// ---- POUs/StringHelper/cutStrNumberToSeperator.TcPOU
{attribute 'no_check'}
//Cut "number" from left site of string. Value will be written into LREAL Target variable in case found string is a valid number
//Function return value will be S_OK if a number is found, S_FALSE if string is empty and E_HRESULTADSERR.ERROR in case found characters are not a number
//Attention! do not use variables smaller then T_MaxString for Source parameter
FUNCTION cutStrNumberToSeperator : HRESULT
VAR_INPUT
	Seperator									:	STRING(5);
END_VAR
VAR_IN_OUT
	Source										:	T_MAXSTRING;
	Target										:	LREAL;
END_VAR
VAR
	tmpString									:	STRING;
	pSource										:	POINTER TO 	T_MAXSTRING;
END_VAR


	pSource										:= ADR(Source);
	tmpString									:= cutStrToSeperator(Seperator, pSource^);
	IF tmpString[0] = 0
	THEN
		cutStrNumberToSeperator					:= S_FALSE;				
	ELSIF isStringNumeric(ADR(tmpString)) 
	THEN 
		Target 									:= TO_LREAL(tmpString); 
	
		cutStrNumberToSeperator					:= S_OK;
	ELSE 
		cutStrNumberToSeperator					:= E_HRESULTADSERR.ERROR;
	END_IF

END_FUNCTION

// ---- POUs/StringHelper/STR_TO_ASC.TcPOU
FUNCTION STR_TO_ASC : BYTE
VAR_INPUT
	str : STRING;
END_VAR
VAR
	pChar : POINTER TO BYTE;
END_VAR

	pChar 		:= ADR(str);
	STR_TO_ASC 	:= pChar^;

END_FUNCTION

// ---- POUs/System/SystemInfo.TcPOU
{attribute 'no_check'}
//Provides all information of PlcAppSystemInfo plus addtional infos like time stamps from various source and in different formats
//
//PlcAppSystemInfo -> https://infosys.beckhoff.com/english.php?content=../content/1033/globaldatatypes/9007199969559691.html&id=7934476013631172214
//TwimCAT time sources -> https://infosys.beckhoff.com/english.php?content=../content/1033/ethercatsystem/2469114379.html&id=
//
FUNCTION_BLOCK SystemInfo
VAR_OUTPUT CONSTANT
{attribute 'displaymode':='binary'}
	OPTION_US_DATE_FORMAT									:	BYTE := 2#0000_0001; //Enable US date format in time stamp - mm/dd/yy
{attribute 'displaymode':='binary'}
	OPTION_US_TIME_FORMAT									:	BYTE := 2#0000_0010; //Enable time in US format - AM/PM vs 24h
{attribute 'displaymode':='binary'} 
	OPTION_TIME_STR_ADD_MS									:	BYTE := 2#0000_0100; //Add ms to time string 
{attribute 'displaymode':='binary'} 
	OPTION_DISABLE_DEV_IDENT								:	BYTE := 2#0000_1000; //Disable to read device identification during boot up (Call FB_GetDeviceIdentificationEx)
END_VAR                     								
VAR_INPUT                   						
	Enable													:	BOOL := TRUE; //Enable function block
	ResetTrig												:	BOOL := FALSE; //Reset Old boot data fault signal
	RtcSyncCylce											:	DWORD := 60; //in seconds - see documentation for "FB_LocalSystemTime"
	KeepOutputsOnBP 										: 	BOOL := FALSE; //The flag can be set to avoid that the outputs are zero-filled if a breakpoint is reached. The task keeps running. Only the execution of PLC code is interrupted.
{attribute 'displaymode':='binary'}
	Options													:	BYTE := 2#0000_0000; //option constants are alreay predefined, so they can accordingly be passed symbolically to the block 
	DateStrSeperator										:	STRING(1) := '/';
END_VAR
VAR_OUTPUT
//PlcAppSystemInfo and cycle time inforamtion from caller task 
	ObjId													: 	OTCID; //Object ID of the PLC project instance
	AdsPort 												: 	UINT; //ADS port of PLC application 
	TComSrvPtr 												: 	ITComObjectServer; // Pointer to TcCOM Object Server 
	AppName													: 	STRING(63); //TwinCAT generated name containing the port number. 
	ProjectName 											: 	STRING(63); //The name of the PLC project. 
	AppTimestampDT											:	DT; //Date and time of application start 
	AppTimestamp											:	STRING(25);	//Date and time of application start in string format
	TaskIndex												:	INT ; //Task index of SysInfo caller
	TaskCnt													: 	UDINT; //The number of tasks in the actual runtime system
	
	Flags 													: 	DWORD; //Boot flags
	LicensesPending 										: 	BOOL;
	BSODOccured 											: 	BOOL;										
	BootDataLoaded											: 	BOOL;//PERSISTENT variables: LOADED (without error)
	OldBootData												: 	BOOL; //PERSISTENT variables: INVALID (the back-up copy was loaded, since no valid data was present)
	NoBootDataLoaded										:	BOOL; //Error no boot data loaded
//	PersistentStatus 										: 	EPlcPersistentStatus;

	LoggedIn												:	BOOL;
	ShutdownInProgress 										: 	BOOL;	
	OnlineChangeCount										: 	UDINT; //The number of online changes made since the last complete download.
	OnlineChange											:	BOOL; //Online change count changed since last plc cycle

{attribute 'displaymode':='hex'}
	CpuCounter												:	ULINT;
	CycleTime         										: 	UDINT;//Cylce time read from PlcAppSystemInfo in multiples of 100 ns.
	CycleTimeNS         									: 	UDINT;//Cylce time in nanoseconds
	CycleTimeT       										: 	TIME; //Cycle time in time format
	CycleTimeLT       										: 	LTIME; //Cycle time in ltime format
	CycleTimeFloat											:	LREAL;//Cycle time in float format <s.ms>

	DevIdentValid											:	BOOL;
	pDevIdent												:	POINTER TO ST_DeviceIdentificationEx := ADR(InstGetDevIdent.stDevIdent);
	
//General	
	TimezoneId												: 	E_TimeZoneID;
	TimeZoneInfo											:	ST_TimeZoneInformation; //Provides actual time zone and bias from local time to UTC e.g. UTC=MEC-01:00 (-60min from lcoal MEZ in Standard time to UTC)
	MonthDays												:	WORD;
	LeapYear												:	BOOL;
	DayOfYear												:	WORD;
	WeekOfYear												:	WORD;
	UtcTimeFT												:	Tc2_Utilities.T_FILETIME; //Current UTC System/TwinCAT time T_FILETIME format, structure representing a 64-bit value with the a number of 100-nanosecond intervals since January 1, 1601 (UTC) (dwLowDateTime : DWORD / dwHighDateTime : DWORD)
//	UtcTimeFT												:	Tc2_Utilities.T_FILETIME64; //Current UTC System/TwinCAT time T_FILETIME format, structure representing a 64-bit value with the a number of 100-nanosecond intervals since January 1, 1601 (UTC) (dwLowDateTime : DWORD / dwHighDateTime : DWORD)
	UtcTimeSTRUCT											:	Tc2_Utilities.TIMESTRUCT; //Current UTC System/TwinCAT time in TIMESTRUCT format
	UtcTimezoneBias											:	DINT;   //Bias from UTC to local time in minutes e.g. MEZ=UTC+01:00 (60min)  
	TimeDT													:	DATE_AND_TIME;	//Current time in DATE_AND_TIME format: DT#1970-01-01-00:00 -> DT#2106-02-06-06:28:15
//	TimeLDT													:	LDATE_AND_TIME;	//Current time in 64bit LDATE_AND_TIME format: DT#1970-01-01-00:00 -> DT#2262-4-10-23:59:59.99999999
	TimeTOD													:	TOD; //Current time in TOD format, range from TOD#00:00 -> TOD#1193:02:47.295
	TimeFT													:	Tc2_Utilities.T_FILETIME; //Current time in T_FILETIME format, structur representing a 64-bit value with the a number of 100-nanosecond intervals since January 1, 1601 (UTC) (dwLowDateTime : DWORD / dwHighDateTime : DWORD)
//	TimeFT													:	Tc2_Utilities.T_FILETIME64; //Current time in T_FILETIME format, structur representing a 64-bit value with the a number of 100-nanosecond intervals since January 1, 1601 (UTC) (dwLowDateTime : DWORD / dwHighDateTime : DWORD)
	TimeSTRUCT												:	Tc2_Utilities.TIMESTRUCT; //Current time in TIMESTRUCT format
	Datestamp												:	DATE; //D#1970-01-01 -> D#2106-02-06
	DateStr													:	STRING(15);	(* dd.mm.jj or mm.dd.jj *)	
	TimeStr													:	STRING(15);	(* hh:mm:ss.xxx or hh:mm:ss.xxxPM/AM *)
	TimeStamp												:	STRING(25); (* DateStr + TimeStr *)	
	TimeStamp2												:	STRING(25); (* YYYY-MM-DDTHHMMSS for example YYYY-MM-DD_HHMMSS_Name.txt *)
	TimeStamp3												:	STRING(25); (* YYYY-MM-DD-hh:mm:ss.xxx *)
	DateStrISO												:	STRING(15);	(* jjjj-mm-dd *)
	TimeStrISO												:	STRING(15);	(* hh:mm:ss *)
	TimeStrISO2												:	STRING(15);	(* hh:mm:ss.xxx *)	
	TimeStampIso											:	STRING(30);	(* jjjj-mm-dd'T'hh:mm:ss.xxx local time*)	
//	TimeStampIsoZulu										:	STRING(30);	(* jjjj-mm-dd'T'hh:mm:ss.xmsZ - Iso timestamp in UTC (ZULU)*)	
//	TimeStampIsoUtc											:	STRING(30);	(* jjjj-mm-dd'T'hh:mm:ss.xms+mm:ss - Iso timestamp with UTC offset *)	

	TimeStampStartup										:	DATE_AND_TIME; //Timestamp of startup
	DCTime													:	Tc2_EtherCAT.T_DCTIME64; //Current TwinCAT distributed clock time in 64-bit T_DCTIME64 format. The smallest unit is a nanosecond.
	DCTimeSTRUCT											:	Tc2_Utilities.TIMESTRUCT;//Current TwinCAT distributed clock time in TIMESTRUCT format
//	SysTimeFT												:	Tc2_Utilities.T_FILETIME64; //Current UTC System/TwinCAT time T_FILETIME format, structure representing a 64-bit value with the a number of 100-nanosecond intervals since January 1, 1601 (UTC) (dwLowDateTime : DWORD / dwHighDateTime : DWORD)
	SysTimeFT												:	Tc2_Utilities.T_FILETIME; //Current UTC System/TwinCAT time T_FILETIME format, structure representing a 32-bit value since January 1, 1601 (UTC) (dwLowDateTime : DWORD / dwHighDateTime : DWORD)
	SysTimeSTRUCT											:	Tc2_Utilities.TIMESTRUCT; //Current UTC System/TwinCAT time in TIMESTRUCT format
	
END_VAR
VAR
	(* Inst. Get Taskindex *)
	InstGETCURTASKINDEX										: 	GETCURTASKINDEX;
	InstLocalSystemTime										:	FB_LocalSystemTime;
	InstNtSetLocalTime										:	NT_SetLocalTime := (NETID := '', TMOUT := DEFAULT_ADS_TIMEOUT);
	InstTimeZoneInfo										:	FB_GetTimeZoneInformation;
	InstCpuCouter											:	GETCPUCOUNTER;
	InstSystemTime											:	GetSystemTime;
	
	
	InstGetDevIdent											:	FB_GetDeviceIdentificationEx;
	_OnlineChangeCount										: 	UDINT; 
	_sec													:	WORD;
	_hour													:	WORD;
	_day													:	WORD;
	_Init													:	BOOL;
END_VAR

	(* Evaluate the PlcAppSystemInfo and and get sytstem timestamp					*)
	(********************************************************************************)
	
(* Get Current Task Index ************************************************************************)
	IF InstGETCURTASKINDEX.index = 0 then InstGETCURTASKINDEX(index => TaskIndex); END_IF

(* Read System Info Current Task *****************************************************************)	
	(* Get static information and boot error messages *)
	IF TwinCAT_SystemInfoVarList._TaskInfo[InstGETCURTASKINDEX.Index].FirstCycle 
	THEN
		AppTimestampDT										:= TwinCAT_SystemInfoVarList._AppInfo.AppTimestamp;
		AppTimestamp										:= DT_TO_STRING(AppTimestampDT);
		AppTimestamp										:= DELETE(AppTimestamp,3,1);
			
		TaskIndex											:= InstGETCURTASKINDEX.Index;
		TaskCnt 											:= TwinCAT_SystemInfoVarList._AppInfo.TaskCnt;
		
		ObjId												:= TwinCAT_SystemInfoVarList._AppInfo.ObjId;
		AppName												:= TwinCAT_SystemInfoVarList._AppInfo.AppName;	
		ProjectName											:= TwinCAT_SystemInfoVarList._AppInfo.ProjectName;	
		AdsPort												:= TwinCAT_SystemInfoVarList._AppInfo.AdsPort;	
			
		Flags												:= TwinCAT_SystemInfoVarList._AppInfo.Flags;
//		PersistentStatus									:= TwinCAT_SystemInfoVarList._AppInfo.PersistentStatus;
		
		BootDataLoaded										:= TwinCAT_SystemInfoVarList._AppInfo.BootDataLoaded;
		OldBootData											:= TwinCAT_SystemInfoVarList._AppInfo.OldBootData;
		NoBootDataLoaded									:= NOT BootDataLoaded AND NOT OldBootData;
		BSODOccured 										:= TwinCAT_SystemInfoVarList._AppInfo.BSODOccured;
		
		CycleTime         									:= TwinCAT_SystemInfoVarList._TaskInfo[TaskIndex].CycleTime;
		CycleTimeNS         								:= TwinCAT_SystemInfoVarList._TaskInfo[TaskIndex].CycleTime * 100;
		CycleTimeT											:= LREAL_TO_TIME(UDINT_TO_LREAL(CycleTime) * 0.0001 );
		CycleTimeLT											:= TO_LTIME(CycleTimeNS);	
		CycleTimeFloat										:= (UDINT_TO_LREAL(CycleTime) * 0.0001 / 1000.0);	
		
	ELSIF ResetTrig
	THEN
		resetBootInfo();
	ELSIF NOT Enable
	THEN
		RETURN;
	END_IF
	
	OnlineChangeCount										:= TwinCAT_SystemInfoVarList._AppInfo.OnlineChangeCnt;
	OnlineChange											:= _OnlineChangeCount <> OnlineChangeCount;
	_OnlineChangeCount										:= OnlineChangeCount;
	LoggedIn 												:= TwinCAT_SystemInfoVarList._AppInfo.LoggedIn;
	ShutdownInProgress 										:= TwinCAT_SystemInfoVarList._AppInfo.ShutdownInProgress;
	LicensesPending 										:= TwinCAT_SystemInfoVarList._AppInfo.LicensesPending;
	TComSrvPtr												:= TwinCAT_SystemInfoVarList._AppInfo.TComSrvPtr;
	TwinCAT_SystemInfoVarList._AppInfo.KeepOutputsOnBP		:= KeepOutputsOnBP;		

(* CPU System counter ****************************************************************************)
	InstCpuCouter(cpuCntLoDW => CpuCounter);	
	MEMCPY(ADR(CpuCounter) + SIZEOF(InstCpuCouter.cpuCntHiDW),ADR(InstCpuCouter.cpuCntHiDW),SIZEOF(InstCpuCouter.cpuCntHiDW));
	
(* Get device identification structure ***********************************************************)
	InstGetDevIdent(
		bExecute	:= NOT Options.3, 
		tTimeout	:= , 
		sNetId		:= , 
		bBusy		=> , 
		bError		=> , 
		nErrorID	=> , 
		stDevIdent	=> );	
	pDevIdent												:= ADR(InstGetDevIdent.stDevIdent);
	IF NOT InstGetDevIdent.bBusy
	THEN
		DevIdentValid										:= NOT InstGetDevIdent.bError;
		
		IF InstGetDevIdent.bError AND ResetTrig
		THEN
			InstGetDevIdent(bExecute := FALSE);			
		END_IF
	ELSE	
		DevIdentValid										:= FALSE;
	END_IF
	
(* Read timezone information every day time ******************************************************)
	IF Enable AND NOT InstTimeZoneInfo.bExecute
		OR InstTimeZoneInfo.bBusy
	THEN
		InstTimeZoneInfo(
			sNetID	:= , 
			bExecute:= TRUE, 
			tTimeout:= , 
			bBusy	=> , 
			bError	=> , 
			nErrID	=> , 
			tzID	=> TimeZoneId, 
			tzInfo	=> TimeZoneInfo);
		IF NOT InstTimeZoneInfo.bBusy 
		THEN
			CASE TimeZoneId OF 
			eTimeZoneID_Invalid:	UtcTimezoneBias			:= 0;				
			eTimeZoneID_Standard:	UtcTimezoneBias			:= -1 * (TimeZoneInfo.bias + TimeZoneInfo.standardBias);
			eTimeZoneID_Daylight:	UtcTimezoneBias			:= -1 * (TimeZoneInfo.bias + TimeZoneInfo.daylightBias);
			ELSE //eTimeZoneID_Unknown:		
				UtcTimezoneBias								:= 0;	
			END_CASE
		END_IF
	ELSIF NOT Enable AND InstTimeZoneInfo.bExecute 
		OR InstTimeZoneInfo.bError AND ResetTrig
	THEN
		InstTimeZoneInfo(bExecute:= FALSE);
	END_IF
		
(* Actual EtherCAT DC time in DCTIME64 format ****************************************************************)
	DCTime													:= F_GetActualDcTime64();
	DCTimeSTRUCT											:= DCTIME64_TO_SYSTEMTIME(DCTime);

(* Get TwinCAT/system time according to system time zone initialized during TC start ******************************************************)
	InstSystemTime(timeHiDW => UtcTimeFT.dwHighDateTime,timeLoDW => UtcTimeFT.dwLowDateTime );
	SysTimeSTRUCT											:= FILETIME_TO_SYSTEMTIME(UTCTimeFT);	
	
//	SysTimeFT												:= F_GetSystemTime();	 
//	SysTimeSTRUCT											:= FILETIME64_TO_SYSTEMTIME(UTCTimeFT);	 
	
(* evalutate systemtime ************************************************************************)
	InstLocalSystemTime(
		sNetID		:= '',
		bEnable		:= Enable,
		dwCycle		:= SEL(InstNtSetLocalTime.START, RtcSyncCylce, 1), //Short update cylce to read windows time after it was set
		dwopt		:= (* Default *),
		tTimeout	:= (* Default *),
		bValid		=> ,
		systemTime	=> TimeSTRUCT,
		tzID		=> );

(* Get TwinCAT/system time in UTC Filetime format ******************************************************)
	IF InstLocalSystemTime.bValid 
	THEN				
		//Update cyclic
//		TimeFT												:= SYSTEMTIME_TO_FILETIME64(TimeSTRUCT);
		TimeFT												:= SYSTEMTIME_TO_FILETIME(TimeSTRUCT);
		TimeDT 												:= SYSTEMTIME_TO_DT(TimeSTRUCT);
//		TimeLDT												:= SYSTEMTIME_TO_LDT(TimeSTRUCT);	
		TimeStamp3											:= SYSTEMTIME_TO_STRING(TimeSTRUCT);
		TimeTOD												:= SEL(Options.2 ,TO_TOD(TimeDT)  , DWORD_TO_TOD(TO_DWORD(TO_TOD(TimeDT)) + TimeSTRUCT.wMilliseconds));  
		TimeStrISO											:= DELETE(TO_STRING(TimeTOD),4,1);

		IF TimeSTRUCT.wMilliseconds < 10 
		THEN
			TimeStrISO2 									:= CONCAT(TimeStrISO,CONCAT('.00',WORD_TO_STRING(TimeSTRUCT.wMilliseconds)));
		ELSIF TimeSTRUCT.wMilliseconds < 100
		THEN
			TimeStrISO2 									:= CONCAT(TimeStrISO,CONCAT('.0',WORD_TO_STRING(TimeSTRUCT.wMilliseconds)));			
		ELSE        										
			TimeStrISO2 									:= CONCAT(TimeStrISO,CONCAT('.',WORD_TO_STRING(TimeSTRUCT.wMilliseconds)));	
		END_IF 	
		
		TimeStampISO										:= CONCAT(DateStrISO , CONCAT('T',TimeStrISO2));
				
		UtcTimeFT											:= F_TranslateFileTimeBias(TimeFT,UtcTimezoneBias,TRUE);
		UtcTimeSTRUCT										:= FILETIME_TO_SYSTEMTIME(UTCTimeFT);	
//		UtcTimeFT											:= F_TranslateFileTime64Bias(TimeFT,UtcTimezoneBias,TRUE);
//		UtcTimeSTRUCT										:= FILETIME64_TO_SYSTEMTIME(UTCTimeFT);	

//		TimeStampIsoZulu									:= SYSTEMTIME_TO_ISO8601(UtcTimeSTRUCT,0,FALSE,3);
//		TimeStampIsoZulu									:= CONCAT(DELETE(TimeStampIsoZulu,6,24),'Z');
//		TimeStampIsoUtc										:= SYSTEMTIME_TO_ISO8601(UtcTimeSTRUCT,TO_INT(UtcTimezoneBias),TRUE,3);
	
		//Create time format
		IF Options.1
		THEN (* US time format hh.mm.ss AM/PM ***************)
			IF TimeSTRUCT.wHour < 10 
			THEN
				TimeStr 									:= CONCAT('0',WORD_TO_STRING(TimeSTRUCT.wHour));
			ELSIF TimeSTRUCT.wHour > 12 
			THEN
				TimeStr 									:= WORD_TO_STRING(TimeSTRUCT.wHour - 12);
				IF TimeSTRUCT.wHour - 12 < 10
				THEN
					TimeStr									:= CONCAT('0',TimeStr);
				END_IF
			ELSE         									
				TimeStr 									:= WORD_TO_STRING(TimeSTRUCT.wHour);
			END_IF		                                    
		ELSE  (* Time hh.mm.ss.xxms ***************)          
			IF TimeSTRUCT.wHour < 10                        
			THEN                                            
				TimeStr 									:= CONCAT('0',WORD_TO_STRING(TimeSTRUCT.wHour));
			ELSE        									
				TimeStr 									:= WORD_TO_STRING(TimeSTRUCT.wHour);
			END_IF			
		END_IF
		
		TimeStr 											:= CONCAT(TimeStr,':');
		
		IF TimeSTRUCT.wMinute < 10 
		THEN
			TimeStr 										:= CONCAT(TimeStr,CONCAT('0',WORD_TO_STRING(TimeSTRUCT.wMinute)));
		ELSE
			TimeStr 										:= CONCAT(TimeStr,WORD_TO_STRING(TimeSTRUCT.wMinute));
		END_IF
		
		TimeStr 											:= CONCAT(TimeStr,':');
		
		IF TimeSTRUCT.wSecond < 10 
		THEN
			TimeStr 										:= CONCAT(TimeStr,CONCAT('0',WORD_TO_STRING(TimeSTRUCT.wSecond)));
		ELSE        										
			TimeStr 										:= CONCAT(TimeStr,WORD_TO_STRING(TimeSTRUCT.wSecond));
		END_IF  
												
		IF Options.2
		THEN //add ms to timestamp
			TimeStr 										:= CONCAT(TimeStr,'.');
			TimeStr 										:= CONCAT(TimeStr,WORD_TO_STRING(TimeSTRUCT.wMilliseconds));
		END_IF
		
		IF Options.1
		THEN //US time format
			TimeStr 										:= CONCAT(TimeStr,SEL(TimeSTRUCT.wHour > 12,' AM', ' PM'));
		END_IF
		
		(* TimeStamp Format DE: DD.MM.YY-Stunde:Minute:Sekunde.xxx,*)
		TimeStamp 											:= CONCAT(DateStr,'-');
		TimeStamp 											:= CONCAT(TimeStamp,TimeStr);
		
		IF _hour <> TimeSTRUCT.wHour OR NOT _Init
		THEN
			_Hour											:= TimeSTRUCT.wHour;		
			//Create date in US fromat with seperator / ************************************************
			IF Options.0
			THEN (* Date mm/dd/jj ********************)
				IF TimeSTRUCT.wMonth < 10 
				THEN
					DateStr 								:= CONCAT('0',WORD_TO_STRING(TimeSTRUCT.wMonth));
				ELSE        								
					DateStr 								:= WORD_TO_STRING(TimeSTRUCT.wMonth);
				END_IF		                                
				DateStr 									:= CONCAT(DateStr,DateStrSeperator);
				IF TimeSTRUCT.wDay < 10                     
				THEN                                        
					DateStr 								:= CONCAT(DateStr,CONCAT('0',WORD_TO_STRING(TimeSTRUCT.wDay)));
				ELSE        								
					DateStr 								:= CONCAT(DateStr,WORD_TO_STRING(TimeSTRUCT.wDay));
				END_IF                                      
															
				DateStr 									:= CONCAT(DateStr,DateStrSeperator);
				DateStr 									:= CONCAT(DateStr,RIGHT(WORD_TO_STRING(TimeSTRUCT.wYear),2));		
		                                                    
			ELSE (* Date dd.mm.jj ********************)	    
				IF TimeSTRUCT.wDay < 10                     
				THEN                                        
					DateStr 								:= CONCAT('0',WORD_TO_STRING(TimeSTRUCT.wDay));
				ELSE        								
					DateStr 								:= WORD_TO_STRING(TimeSTRUCT.wDay);
				END_IF                                      
				DateStr 									:= CONCAT(DateStr,DateStrSeperator);
				IF TimeSTRUCT.wMonth < 10                   
				THEN                                        
					DateStr 								:= CONCAT(DateStr,CONCAT('0',WORD_TO_STRING(TimeSTRUCT.wMonth)));
				ELSE        								
					DateStr 								:= CONCAT(DateStr,WORD_TO_STRING(TimeSTRUCT.wMonth));
				END_IF                                      
															
				DateStr 									:= CONCAT(DateStr,DateStrSeperator);
				DateStr 									:= CONCAT(DateStr,RIGHT(WORD_TO_STRING(TimeSTRUCT.wYear),2));	
			END_IF      

			DateStrISO										:= DELETE(TO_STRING(TO_DATE(TimeDT)),2,1);
			
			(* information of year *)                       
			MonthDays										:= F_GetMaxMonthDays(TimeSTRUCT.wYear,TimeSTRUCT.wMonth);
			LeapYear										:= F_YearIsLeapYear(TimeSTRUCT.wYear) ;
			WeekOfYear										:= F_GetWeekOfTheYear(TimeDT);
			DayOfYear										:= F_GetDOYOfYearMonthDay(TimeSTRUCT.wYear,TimeSTRUCT.wMonth,TimeSTRUCT.wDay);
			DateStamp										:= TO_DATE(TimeDT);		
			
			IF NOT _INIT AND_THEN TO_DINT(TimeStampStartup) = 0  
			THEN					
				TimeStampStartup							:= SYSTEMTIME_TO_DT(TimeSTRUCT);
			END_IF
			
			IF NOT InstTimeZoneInfo.bBusy THEN InstTimeZoneInfo(bExecute:= FALSE); END_IF

            _INIT											:= TRUE;            
		END_IF //hour
		
		IF _sec <> TimeSTRUCT.wSecond 
		THEN	
			_sec 											:= TimeSTRUCT.wSecond;
														
			(* TimeStamp2 FileName YYYY-MM-DD_HHMMSS *)
			TimeStamp2										:= CONCAT(DateStrISO , '_');
			IF TimeSTRUCT.wHour < 10                    	
			THEN                                        	
				TimeStamp2 									:= CONCAT(TimeStamp2,CONCAT('0',WORD_TO_STRING(TimeSTRUCT.wHour)));
			ELSE           									
				TimeStamp2 									:= CONCAT(TimeStamp2,WORD_TO_STRING(TimeSTRUCT.wHour));
			END_IF                                      	
			IF TimeSTRUCT.wMinute < 10                  	
			THEN                                        	
				TimeStamp2 									:= CONCAT(TimeStamp2,CONCAT('0',WORD_TO_STRING(TimeSTRUCT.wMinute)));
			ELSE           									
				TimeStamp2 									:= CONCAT(TimeStamp2,WORD_TO_STRING(TimeSTRUCT.wMinute));
			END_IF                                      	
			IF TimeSTRUCT.wSecond < 10                  	
			THEN                                        	
				TimeStamp2 									:= CONCAT(TimeStamp2,CONCAT('0',WORD_TO_STRING(TimeSTRUCT.wSecond)));
			ELSE           									
				TimeStamp2 									:= CONCAT(TimeStamp2,WORD_TO_STRING(TimeSTRUCT.wSecond));
			END_IF
		END_IF //second update
													
	END_IF

(* set system time *****************************************************************************)
	InstNtSetLocalTime(
		NETID		:= , 
		TIMESTR		:= , 
		START		:= , // Start by Methode "SetSysTime" 
		TMOUT		:= , 
		BUSY		=> , 
		ERR			=> ); 
	
	IF InstNtSetLocalTime.START AND NOT InstNtSetLocalTime.BUSY
	THEN //Take care that all timestamp get updated after set a new time
		InstNtSetLocalTime.START							:= FALSE;	
		_Init												:= FALSE;								
	END_IF
	
(**************************************************************************************************)

PROPERTY PUBLIC actDCTimeWithTimezoneBias : T_DCTIME64
GET
actDCTimeWithTimezoneBias							:= F_GetActualDcTime64() + (TO_ULINT(UtcTimezoneBias) * 60 * EC_DCTIME_TICKSPERSEC64);
END_GET
END_PROPERTY

PROPERTY PUBLIC optAddmsToTimeString : BOOL
GET
optAddmsToTimeString := Options.2;
END_GET
SET
Options.2 := optAddmsToTimeString;
END_SET
END_PROPERTY

PROPERTY PUBLIC  optDisableReadDeviceIdentification : BOOL
GET
optDisableReadDeviceIdentification := Options.3;
END_GET
SET
Options.3 := optDisableReadDeviceIdentification;
END_SET
END_PROPERTY

PROPERTY PUBLIC optEnableUSDateFormat : BOOL
GET
optEnableUSDateFormat := Options.0;
END_GET
SET
Options.0 := optEnableUSDateFormat;
END_SET
END_PROPERTY

PROPERTY PUBLIC optEnableUSTimeFormat : BOOL
GET
optEnableUSTimeFormat := Options.1;
END_GET
SET
Options.1 := optEnableUSTimeFormat;
END_SET
END_PROPERTY

METHOD PUBLIC resetBootInfo : BOOL  //Return value = TRUE if execution finished
VAR_INPUT
END_VAR
OldBootData 												:= FALSE;
BSODOccured													:= FALSE;
NoBootDataLoaded											:= FALSE;
resetBootInfo												:= TRUE;
END_METHOD

METHOD PUBLIC setSysTime  : BOOL //Return value = TRUE if execution finished
VAR_INPUT
	TimeStruct		: TIMESTRUCT;
END_VAR
InstNtSetLocalTime(
		NETID		:= '', 
		TIMESTR		:= TimeStruct, 
		START		:= NOT InstNtSetLocalTime.START AND TimeStruct.wYear > 2000 
						AND TimeStruct.wDay > 0 AND TimeStruct.wMonth	< 32	
						AND TimeStruct.wMonth > 0 AND TimeStruct.wMonth	< 13	
						AND TimeStruct.wHour >= 0 AND TimeStruct.wHour	< 24	
						AND TimeStruct.wMinute >= 0 AND TimeStruct.wMinute < 60
						AND TimeStruct.wSecond >= 0 AND TimeStruct.wSecond < 60				
						OR InstNtSetLocalTime.BUSY, 
		TMOUT		:= , 
		BUSY		=> , 
		ERR			=> , 
		ERRID		=> );
		
setSysTime													:= InstNtSetLocalTime.BUSY;
END_METHOD

END_FUNCTION_BLOCK

// ---- POUs/System/SystemInfo64.TcPOU
{attribute 'no_check'}
//Provides all information of PlcAppSystemInfo plus addtional infos like time stamps from various source and in different formats
//
//PlcAppSystemInfo -> https://infosys.beckhoff.com/english.php?content=../content/1033/globaldatatypes/9007199969559691.html&id=7934476013631172214
//TwimCAT time sources -> https://infosys.beckhoff.com/english.php?content=../content/1033/ethercatsystem/2469114379.html&id=
//
FUNCTION_BLOCK SystemInfo64
VAR_OUTPUT CONSTANT
{attribute 'displaymode':='binary'}
	OPTION_US_DATE_FORMAT									:	BYTE := 2#0000_0001; //Enable US date format in time stamp - mm/dd/yy
{attribute 'displaymode':='binary'}
	OPTION_US_TIME_FORMAT									:	BYTE := 2#0000_0010; //Enable time in US format - AM/PM vs 24h
{attribute 'displaymode':='binary'} 
	OPTION_TIME_STR_ADD_MS									:	BYTE := 2#0000_0100; //Add ms to time string 
{attribute 'displaymode':='binary'} 
	OPTION_DISABLE_DEV_IDENT								:	BYTE := 2#0000_1000; //Disable to read device identification during boot up (Call FB_GetDeviceIdentificationEx)
END_VAR                     								
VAR_INPUT                   						
	Enable													:	BOOL := TRUE; //Enable function block
	ResetTrig												:	BOOL := FALSE; //Reset Old boot data fault signal
	RtcSyncCylce											:	DWORD := 60; //in seconds - see documentation for "FB_LocalSystemTime"
	KeepOutputsOnBP 										: 	BOOL := FALSE; //The flag can be set to avoid that the outputs are zero-filled if a breakpoint is reached. The task keeps running. Only the execution of PLC code is interrupted.
{attribute 'displaymode':='binary'}
	Options													:	BYTE := 2#0000_0000; //option constants are alreay predefined, so they can accordingly be passed symbolically to the block 
	DateStrSeperator										:	STRING(1) := '/';
END_VAR
VAR_OUTPUT
//PlcAppSystemInfo and cycle time inforamtion from caller task 
	ObjId													: 	OTCID; //Object ID of the PLC project instance
	AdsPort 												: 	UINT; //ADS port of PLC application 
	TComSrvPtr 												: 	ITComObjectServer; // Pointer to TcCOM Object Server 
	AppName													: 	STRING(63); //TwinCAT generated name containing the port number. 
	ProjectName 											: 	STRING(63); //The name of the PLC project. 
	AppTimestampDT											:	DT; //Date and time of application start 
	AppTimestamp											:	STRING(25);	//Date and time of application start in string format
	TaskIndex												:	INT ; //Task index of SysInfo caller
	TaskCnt													: 	UDINT; //The number of tasks in the actual runtime system
	
	Flags 													: 	DWORD; //Boot flags
	LicensesPending 										: 	BOOL;
	BSODOccured 											: 	BOOL;										
	BootDataLoaded											: 	BOOL;//PERSISTENT variables: LOADED (without error)
	OldBootData												: 	BOOL; //PERSISTENT variables: INVALID (the back-up copy was loaded, since no valid data was present)
	NoBootDataLoaded										:	BOOL; //Error no boot data loaded
//	PersistentStatus 										: 	EPlcPersistentStatus;

	LoggedIn												:	BOOL;
	ShutdownInProgress 										: 	BOOL;	
	OnlineChangeCount										: 	UDINT; //The number of online changes made since the last complete download.
	OnlineChange											:	BOOL; //Online change count changed since last plc cycle

{attribute 'displaymode':='hex'}
	CpuCounter												:	ULINT;
	CycleTime         										: 	UDINT;//Cylce time read from PlcAppSystemInfo in multiples of 100 ns.
	CycleTimeNS         									: 	UDINT;//Cylce time in nanoseconds
	CycleTimeT       										: 	TIME; //Cycle time in time format
	CycleTimeLT       										: 	LTIME; //Cycle time in ltime format
	CycleTimeFloat											:	LREAL;//Cycle time in float format <s.ms>

	DevIdentValid											:	BOOL;
	pDevIdent												:	POINTER TO ST_DeviceIdentificationEx := ADR(InstGetDevIdent.stDevIdent);
	
//General	
	TimezoneId												: 	E_TimeZoneID;
	TimeZoneInfo											:	ST_TimeZoneInformation;
	MonthDays												:	WORD;
	LeapYear												:	BOOL;
	DayOfYear												:	WORD;
	WeekOfYear												:	WORD;
	UtcTimeFT												:	Tc2_Utilities.T_FILETIME64; //Current UTC System/TwinCAT time T_FILETIME format, structure representing a 64-bit value with the a number of 100-nanosecond intervals since January 1, 1601 (UTC) (dwLowDateTime : DWORD / dwHighDateTime : DWORD)
	UtcTimeSTRUCT											:	Tc2_Utilities.TIMESTRUCT; //Current UTC System/TwinCAT time in TIMESTRUCT format
	UtcTimezoneBias											:	DINT;   //Total timezone bias in minutes to UTC 
	TimeDT													:	DATE_AND_TIME;	//Current time in DATE_AND_TIME format: DT#1970-01-01-00:00 -> DT#2106-02-06-06:28:15
//	TimeLDT													:	LDATE_AND_TIME;	//Current time in 64bit LDATE_AND_TIME format: DT#1970-01-01-00:00 -> DT#2262-4-10-23:59:59.99999999
	TimeTOD													:	TOD; //Current time in TOD format, range from TOD#00:00 -> TOD#1193:02:47.295
	TimeFT													:	Tc2_Utilities.T_FILETIME64; //Current time in T_FILETIME format, structur representing a 64-bit value with the a number of 100-nanosecond intervals since January 1, 1601 (UTC) (dwLowDateTime : DWORD / dwHighDateTime : DWORD)
	TimeSTRUCT												:	Tc2_Utilities.TIMESTRUCT; //Current time in TIMESTRUCT format
	Datestamp												:	DATE; //D#1970-01-01 -> D#2106-02-06
	DateStr													:	STRING(15);	(* dd.mm.jj or mm.dd.jj *)	
	TimeStr													:	STRING(15);	(* hh:mm:ss.xxx or hh:mm:ss.xxxPM/AM *)
	TimeStamp												:	STRING(25); (* DateStr + TimeStr *)	
	TimeStamp2												:	STRING(25); (* YYYY-MM-DDTHHMMSS for example YYYY-MM-DD_HHMMSS_Name.txt *)
	TimeStamp3												:	STRING(25); (* YYYY-MM-DD-hh:mm:ss.xxx *)
	DateStrISO												:	STRING(15);	(* jj-mm-dd *)
	TimeStrISO												:	STRING(15);	(* hh:mm:ss *)
	TimeStampISO											:	STRING(25);	(* jj-mm-dd'T'hh:mm:ss.xxms *)	
	TimeStampStartup										:	DATE_AND_TIME; //Timestamp of startup
	DCTime													:	Tc2_EtherCAT.T_DCTIME64; //Current TwinCAT distributed clock time in 64-bit T_DCTIME64 format. The smallest unit is a nanosecond.
	DCTimeSTRUCT											:	Tc2_Utilities.TIMESTRUCT;//Current TwinCAT distributed clock time in TIMESTRUCT format
	SysTimeFT												:	Tc2_Utilities.T_FILETIME64; //Current UTC System/TwinCAT time T_FILETIME format, structure representing a 64-bit value with the a number of 100-nanosecond intervals since January 1, 1601 (UTC) (dwLowDateTime : DWORD / dwHighDateTime : DWORD)
	SysTimeSTRUCT											:	Tc2_Utilities.TIMESTRUCT; //Current UTC System/TwinCAT time in TIMESTRUCT format
	
END_VAR
VAR
	(* Inst. Get Taskindex *)
	InstGETCURTASKINDEX										: 	GETCURTASKINDEX;
	InstLocalSystemTime										:	FB_LocalSystemTime;
	InstNtSetLocalTime										:	NT_SetLocalTime := (NETID := '', TMOUT := DEFAULT_ADS_TIMEOUT);
	InstTimeZoneInfo										:	FB_GetTimeZoneInformation;
	InstCpuCouter											:	GETCPUCOUNTER;
	
	InstGetDevIdent											:	FB_GetDeviceIdentificationEx;
	_OnlineChangeCount										: 	UDINT; 
	_sec													:	WORD;
	_hour													:	WORD;
	_day													:	WORD;
	_Init													:	BOOL;
END_VAR

	(* Evaluate the PlcAppSystemInfo and and get sytstem timestamp					*)
	(********************************************************************************)
	
(* Get Current Task Index ************************************************************************)
	IF InstGETCURTASKINDEX.index = 0 then InstGETCURTASKINDEX(index => TaskIndex); END_IF

(* Read System Info Current Task *****************************************************************)	
	(* Get static information and boot error messages *)
	IF TwinCAT_SystemInfoVarList._TaskInfo[InstGETCURTASKINDEX.Index].FirstCycle 
	THEN
		AppTimestampDT										:= TwinCAT_SystemInfoVarList._AppInfo.AppTimestamp;
		AppTimestamp										:= DT_TO_STRING(AppTimestampDT);
		AppTimestamp										:= DELETE(AppTimestamp,3,1);
			
		TaskIndex											:= InstGETCURTASKINDEX.Index;
		TaskCnt 											:= TwinCAT_SystemInfoVarList._AppInfo.TaskCnt;
		
		ObjId												:= TwinCAT_SystemInfoVarList._AppInfo.ObjId;
		AppName												:= TwinCAT_SystemInfoVarList._AppInfo.AppName;	
		ProjectName											:= TwinCAT_SystemInfoVarList._AppInfo.ProjectName;	
		AdsPort												:= TwinCAT_SystemInfoVarList._AppInfo.AdsPort;	
			
		Flags												:= TwinCAT_SystemInfoVarList._AppInfo.Flags;
//		PersistentStatus									:= TwinCAT_SystemInfoVarList._AppInfo.PersistentStatus;
		
		BootDataLoaded										:= TwinCAT_SystemInfoVarList._AppInfo.BootDataLoaded;
		OldBootData											:= TwinCAT_SystemInfoVarList._AppInfo.OldBootData;
		NoBootDataLoaded									:= NOT BootDataLoaded AND NOT OldBootData;
		BSODOccured 										:= TwinCAT_SystemInfoVarList._AppInfo.BSODOccured;
		
		CycleTime         									:= TwinCAT_SystemInfoVarList._TaskInfo[TaskIndex].CycleTime;
		CycleTimeNS         								:= TwinCAT_SystemInfoVarList._TaskInfo[TaskIndex].CycleTime * 100;
		CycleTimeT											:= LREAL_TO_TIME(UDINT_TO_LREAL(CycleTime) * 0.0001 );
		CycleTimeLT											:= TO_LTIME(CycleTimeNS);	
		CycleTimeFloat										:= (UDINT_TO_LREAL(CycleTime) * 0.0001 / 1000.0);	
		
	ELSIF ResetTrig
	THEN
		resetBootInfo();
	ELSIF NOT Enable
	THEN
		RETURN;
	END_IF
	
	OnlineChangeCount										:= TwinCAT_SystemInfoVarList._AppInfo.OnlineChangeCnt;
	OnlineChange											:= _OnlineChangeCount <> OnlineChangeCount;
	_OnlineChangeCount										:= OnlineChangeCount;
	LoggedIn 												:= TwinCAT_SystemInfoVarList._AppInfo.LoggedIn;
	ShutdownInProgress 										:= TwinCAT_SystemInfoVarList._AppInfo.ShutdownInProgress;
	LicensesPending 										:= TwinCAT_SystemInfoVarList._AppInfo.LicensesPending;
	TComSrvPtr												:= TwinCAT_SystemInfoVarList._AppInfo.TComSrvPtr;
	TwinCAT_SystemInfoVarList._AppInfo.KeepOutputsOnBP		:= KeepOutputsOnBP;		

(* CPU System counter ****************************************************************************)
	InstCpuCouter(cpuCntLoDW => CpuCounter);	
	MEMCPY(ADR(CpuCounter) + SIZEOF(InstCpuCouter.cpuCntHiDW),ADR(InstCpuCouter.cpuCntHiDW),SIZEOF(InstCpuCouter.cpuCntHiDW));
	
(* Get device identification structure ***********************************************************)
	InstGetDevIdent(
		bExecute	:= NOT Options.3, 
		tTimeout	:= , 
		sNetId		:= , 
		bBusy		=> , 
		bError		=> , 
		nErrorID	=> , 
		stDevIdent	=> );	
	pDevIdent												:= ADR(InstGetDevIdent.stDevIdent);
	IF NOT InstGetDevIdent.bBusy
	THEN
		DevIdentValid										:= NOT InstGetDevIdent.bError;
		
		IF InstGetDevIdent.bError AND ResetTrig
		THEN
			InstGetDevIdent(bExecute := FALSE);			
		END_IF
	ELSE	
		DevIdentValid										:= FALSE;
	END_IF
	
(* Read timezone information every day time ******************************************************)
	IF Enable AND NOT InstTimeZoneInfo.bExecute
		OR InstTimeZoneInfo.bBusy
	THEN
		InstTimeZoneInfo(
			sNetID	:= , 
			bExecute:= TRUE, 
			tTimeout:= , 
			bBusy	=> , 
			bError	=> , 
			nErrID	=> , 
			tzID	=> TimeZoneId, 
			tzInfo	=> TimeZoneInfo);
		IF NOT InstTimeZoneInfo.bBusy 
		THEN
			CASE TimeZoneId OF 
			eTimeZoneID_Invalid:	UtcTimezoneBias			:= 0;				
			eTimeZoneID_Standard:	UtcTimezoneBias			:= -1 * (TimeZoneInfo.bias);
			eTimeZoneID_Daylight:	UtcTimezoneBias			:= -1 * (TimeZoneInfo.bias + TimeZoneInfo.daylightBias);
			ELSE //eTimeZoneID_Unknown:		
				UtcTimezoneBias								:= 0;	
			END_CASE
		END_IF
	ELSIF NOT Enable AND InstTimeZoneInfo.bExecute 
		OR InstTimeZoneInfo.bError AND ResetTrig
	THEN
		InstTimeZoneInfo(bExecute:= FALSE);
	END_IF
		
(* Actual EtherCAT DC time in DCTIME64 format ****************************************************************)
	DCTime													:= F_GetActualDcTime64();
	DCTimeSTRUCT											:= DCTIME64_TO_SYSTEMTIME(DCTime);

(* Get TwinCAT/system time according to system time zone initialized during TC start ******************************************************)
	SysTimeFT												:= F_GetSystemTime();	 
	SysTimeSTRUCT											:= FILETIME64_TO_SYSTEMTIME(UTCTimeFT);	 
	
(* evalutate systemtime ************************************************************************)
	InstLocalSystemTime(
		sNetID		:= '',
		bEnable		:= Enable,
		dwCycle		:= SEL(InstNtSetLocalTime.START, RtcSyncCylce, 1), //Short update cylce to read windows time after it was set
		dwopt		:= (* Default *),
		tTimeout	:= (* Default *),
		bValid		=> ,
		systemTime	=> TimeSTRUCT,
		tzID		=> );

(* Get TwinCAT/system time in UTC Filetime format ******************************************************)
	IF InstLocalSystemTime.bValid 
	THEN				
		//Update cyclic
		TimeFT												:= SYSTEMTIME_TO_FILETIME64(TimeSTRUCT);
		TimeDT 												:= SYSTEMTIME_TO_DT(TimeSTRUCT);
//		TimeLDT												:= SYSTEMTIME_TO_LDT(TimeSTRUCT);	
		TimeStamp3											:= SYSTEMTIME_TO_STRING(TimeSTRUCT);
		TimeTOD												:= SEL(Options.2 ,TO_TOD(TimeDT)  , DWORD_TO_TOD(TO_DWORD(TO_TOD(TimeDT)) + TimeSTRUCT.wMilliseconds));  
		TimeStrISO											:= DELETE(TO_STRING(TimeTOD),4,1);
		TimeStampISO										:= CONCAT(DateStrISO , CONCAT('T',TimeStrISO));
		
		UtcTimeFT											:= F_TranslateFileTime64Bias(TimeFT,UtcTimezoneBias,TRUE);
		UtcTimeSTRUCT										:= FILETIME64_TO_SYSTEMTIME(UTCTimeFT);	
	
		//Create time format
		IF Options.1
		THEN (* US time format hh.mm.ss AM/PM ***************)
			IF TimeSTRUCT.wHour < 10 
			THEN
				TimeStr 									:= CONCAT('0',WORD_TO_STRING(TimeSTRUCT.wHour));
			ELSIF TimeSTRUCT.wHour > 12 
			THEN
				TimeStr 									:= WORD_TO_STRING(TimeSTRUCT.wHour - 12);
				IF TimeSTRUCT.wHour - 12 < 10
				THEN
					TimeStr									:= CONCAT('0',TimeStr);
				END_IF
			ELSE         									
				TimeStr 									:= WORD_TO_STRING(TimeSTRUCT.wHour);
			END_IF		                                    
		ELSE  (* Time hh.mm.ss.xxms ***************)          
			IF TimeSTRUCT.wHour < 10                        
			THEN                                            
				TimeStr 									:= CONCAT('0',WORD_TO_STRING(TimeSTRUCT.wHour));
			ELSE        									
				TimeStr 									:= WORD_TO_STRING(TimeSTRUCT.wHour);
			END_IF			
		END_IF
		
		TimeStr 											:= CONCAT(TimeStr,':');
		
		IF TimeSTRUCT.wMinute < 10 
		THEN
			TimeStr 										:= CONCAT(TimeStr,CONCAT('0',WORD_TO_STRING(TimeSTRUCT.wMinute)));
		ELSE
			TimeStr 										:= CONCAT(TimeStr,WORD_TO_STRING(TimeSTRUCT.wMinute));
		END_IF
		
		TimeStr 											:= CONCAT(TimeStr,':');
		
		IF TimeSTRUCT.wSecond < 10 
		THEN
			TimeStr 										:= CONCAT(TimeStr,CONCAT('0',WORD_TO_STRING(TimeSTRUCT.wSecond)));
		ELSE        										
			TimeStr 										:= CONCAT(TimeStr,WORD_TO_STRING(TimeSTRUCT.wSecond));
		END_IF  
												
		IF Options.2
		THEN //add ms to timestamp
			TimeStr 										:= CONCAT(TimeStr,'.');
			TimeStr 										:= CONCAT(TimeStr,WORD_TO_STRING(TimeSTRUCT.wMilliseconds));
		END_IF
		
		IF Options.1
		THEN //US time format
			TimeStr 										:= CONCAT(TimeStr,SEL(TimeSTRUCT.wHour > 12,' AM', ' PM'));
		END_IF
		
		(* TimeStamp Format DE: DD.MM.YY-Stunde:Minute:Sekunde.xxx,*)
		TimeStamp 											:= CONCAT(DateStr,'-');
		TimeStamp 											:= CONCAT(TimeStamp,TimeStr);
		
		IF _hour <> TimeSTRUCT.wHour OR NOT _Init
		THEN
			_Hour											:= TimeSTRUCT.wHour;		
			//Create date in US fromat with seperator / ************************************************
			IF Options.0
			THEN (* Date mm/dd/jj ********************)
				IF TimeSTRUCT.wMonth < 10 
				THEN
					DateStr 								:= CONCAT('0',WORD_TO_STRING(TimeSTRUCT.wMonth));
				ELSE        								
					DateStr 								:= WORD_TO_STRING(TimeSTRUCT.wMonth);
				END_IF		                                
				DateStr 									:= CONCAT(DateStr,DateStrSeperator);
				IF TimeSTRUCT.wDay < 10                     
				THEN                                        
					DateStr 								:= CONCAT(DateStr,CONCAT('0',WORD_TO_STRING(TimeSTRUCT.wDay)));
				ELSE        								
					DateStr 								:= CONCAT(DateStr,WORD_TO_STRING(TimeSTRUCT.wDay));
				END_IF                                      
															
				DateStr 									:= CONCAT(DateStr,DateStrSeperator);
				DateStr 									:= CONCAT(DateStr,RIGHT(WORD_TO_STRING(TimeSTRUCT.wYear),2));		
		                                                    
			ELSE (* Date dd.mm.jj ********************)	    
				IF TimeSTRUCT.wDay < 10                     
				THEN                                        
					DateStr 								:= CONCAT('0',WORD_TO_STRING(TimeSTRUCT.wDay));
				ELSE        								
					DateStr 								:= WORD_TO_STRING(TimeSTRUCT.wDay);
				END_IF                                      
				DateStr 									:= CONCAT(DateStr,DateStrSeperator);
				IF TimeSTRUCT.wMonth < 10                   
				THEN                                        
					DateStr 								:= CONCAT(DateStr,CONCAT('0',WORD_TO_STRING(TimeSTRUCT.wMonth)));
				ELSE        								
					DateStr 								:= CONCAT(DateStr,WORD_TO_STRING(TimeSTRUCT.wMonth));
				END_IF                                      
															
				DateStr 									:= CONCAT(DateStr,DateStrSeperator);
				DateStr 									:= CONCAT(DateStr,RIGHT(WORD_TO_STRING(TimeSTRUCT.wYear),2));	
			END_IF      

			DateStrISO										:= DELETE(TO_STRING(TO_DATE(TimeDT)),2,1);
			
			(* information of year *)                       
			MonthDays										:= F_GetMaxMonthDays(TimeSTRUCT.wYear,TimeSTRUCT.wMonth);
			LeapYear										:= F_YearIsLeapYear(TimeSTRUCT.wYear) ;
			WeekOfYear										:= F_GetWeekOfTheYear(TimeDT);
			DayOfYear										:= F_GetDOYOfYearMonthDay(TimeSTRUCT.wYear,TimeSTRUCT.wMonth,TimeSTRUCT.wDay);
			DateStamp										:= TO_DATE(TimeDT);		
			
			IF NOT _INIT AND_THEN TO_DINT(TimeStampStartup) = 0  
			THEN					
				TimeStampStartup							:= SYSTEMTIME_TO_DT(TimeSTRUCT);
			END_IF
			
			IF NOT InstTimeZoneInfo.bBusy THEN InstTimeZoneInfo(bExecute:= FALSE); END_IF

            _INIT											:= TRUE;            
		END_IF //hour
		
		IF _sec <> TimeSTRUCT.wSecond 
		THEN	
			_sec 											:= TimeSTRUCT.wSecond;
														
			(* TimeStamp2 FileName YYYY-MM-DD_HHMMSS *)
			TimeStamp2										:= CONCAT(DateStrISO , '_');
			IF TimeSTRUCT.wHour < 10                    	
			THEN                                        	
				TimeStamp2 									:= CONCAT(TimeStamp2,CONCAT('0',WORD_TO_STRING(TimeSTRUCT.wHour)));
			ELSE           									
				TimeStamp2 									:= CONCAT(TimeStamp2,WORD_TO_STRING(TimeSTRUCT.wHour));
			END_IF                                      	
			IF TimeSTRUCT.wMinute < 10                  	
			THEN                                        	
				TimeStamp2 									:= CONCAT(TimeStamp2,CONCAT('0',WORD_TO_STRING(TimeSTRUCT.wMinute)));
			ELSE           									
				TimeStamp2 									:= CONCAT(TimeStamp2,WORD_TO_STRING(TimeSTRUCT.wMinute));
			END_IF                                      	
			IF TimeSTRUCT.wSecond < 10                  	
			THEN                                        	
				TimeStamp2 									:= CONCAT(TimeStamp2,CONCAT('0',WORD_TO_STRING(TimeSTRUCT.wSecond)));
			ELSE           									
				TimeStamp2 									:= CONCAT(TimeStamp2,WORD_TO_STRING(TimeSTRUCT.wSecond));
			END_IF
		END_IF //second update
													
	END_IF

(* set system time *****************************************************************************)
	InstNtSetLocalTime(
		NETID		:= , 
		TIMESTR		:= , 
		START		:= , // Start by Methode "SetSysTime" 
		TMOUT		:= , 
		BUSY		=> , 
		ERR			=> ); 
	
	IF InstNtSetLocalTime.START AND NOT InstNtSetLocalTime.BUSY
	THEN //Take care that all timestamp get updated after set a new time
		InstNtSetLocalTime.START							:= FALSE;	
		_Init												:= FALSE;								
	END_IF
	
(**************************************************************************************************)

PROPERTY PUBLIC actDCTimeWithTimezoneBias : T_DCTIME64
GET
actDCTimeWithTimezoneBias							:= F_GetActualDcTime64() + (TO_ULINT(UtcTimezoneBias) * 60 * EC_DCTIME_TICKSPERSEC64);
END_GET
END_PROPERTY

PROPERTY PUBLIC actSysTimeWithTimezoneBias : T_FILETIME64
GET
actSysTimeWithTimezoneBias							:= F_GetSystemTime() + (TO_ULINT(UtcTimezoneBias) * 60 * EC_DCTIME_TICKSPERSEC64);
END_GET
END_PROPERTY

PROPERTY PUBLIC optAddmsToTimeString : BOOL
GET
optAddmsToTimeString := Options.2;
END_GET
SET
Options.2 := optAddmsToTimeString;
END_SET
END_PROPERTY

PROPERTY PUBLIC  optDisableReadDeviceIdentification : BOOL
GET
optDisableReadDeviceIdentification := Options.3;
END_GET
SET
Options.3 := optDisableReadDeviceIdentification;
END_SET
END_PROPERTY

PROPERTY PUBLIC optEnableUSDateFormat : BOOL
GET
optEnableUSDateFormat := Options.0;
END_GET
SET
Options.0 := optEnableUSDateFormat;
END_SET
END_PROPERTY

PROPERTY PUBLIC optEnableUSTimeFormat : BOOL
GET
optEnableUSTimeFormat := Options.1;
END_GET
SET
Options.1 := optEnableUSTimeFormat;
END_SET
END_PROPERTY

METHOD PUBLIC resetBootInfo : BOOL  //Return value = TRUE if execution finished
VAR_INPUT
END_VAR
OldBootData 												:= FALSE;
BSODOccured													:= FALSE;
NoBootDataLoaded											:= FALSE;
resetBootInfo												:= TRUE;
END_METHOD

METHOD PUBLIC setSysTime  : BOOL //Return value = TRUE if execution finished
VAR_INPUT
	TimeStruct		: TIMESTRUCT;
END_VAR
InstNtSetLocalTime(
		NETID		:= '', 
		TIMESTR		:= TimeStruct, 
		START		:= NOT InstNtSetLocalTime.START AND TimeStruct.wYear > 2000 
						AND TimeStruct.wDay > 0 AND TimeStruct.wMonth	< 32	
						AND TimeStruct.wMonth > 0 AND TimeStruct.wMonth	< 13	
						AND TimeStruct.wHour >= 0 AND TimeStruct.wHour	< 24	
						AND TimeStruct.wMinute >= 0 AND TimeStruct.wMinute < 60
						AND TimeStruct.wSecond >= 0 AND TimeStruct.wSecond < 60				
						OR InstNtSetLocalTime.BUSY, 
		TMOUT		:= , 
		BUSY		=> , 
		ERR			=> , 
		ERRID		=> );
		
setSysTime													:= InstNtSetLocalTime.BUSY;
END_METHOD

END_FUNCTION_BLOCK

// ---- POUs/TimeHelper/PartsPerTime.TcPOU
{attribute 'no_check'}
//This function-block counts pieces/parts per selectable basetime 
FUNCTION_BLOCK PartsPerTime
VAR_INPUT
	NewPartTrig												: 	BOOL	:= FALSE;	// event
	ResetTrig												: 	BOOL	:= FALSE;	// reset counter
	Basetime												:	TIME 	:= T#60S;	// basetime
END_VAR             										
VAR_OUTPUT          										
	Forecast												: 	LREAL;				// calulated forecast for basetime
	Counted													: 	DINT;				// counted impulses in last basetime period
	CountAct												:	DINT;				// actual counter in basetime period
	Q_RT													:	BOOL;				// rising event of trigger input
END_VAR             										
VAR                 										
	rtTrigger												: 	R_TRIG;
	TON														:	TON;
	StartTime												: 	TIME;
	StartTime_Old											: 	TIME;
	TimeImpImp												: 	TIME;
END_VAR

rtTrigger(CLK := NewPartTrig,Q => Q_RT);
TON(IN := NOT TON.Q AND NOT ResetTrig, PT := Basetime);

IF TON.Q 
THEN
	Counted 												:= CountAct;
	CountAct 												:= 0;
END_IF

IF ResetTrig 
THEN
	reset();
ELSIF rtTrigger.Q 
THEN
	addNewPart();
END_IF

METHOD PUBLIC addNewPart : BOOL //Return value = TRUE if execution finished
VAR_INPUT
END_VAR
	StartTime_Old 											:= StartTime;
	StartTime 												:= TIME();
	TimeImpImp	 											:= MAX(T#1MS ,StartTime - StartTime_Old);
	Forecast	 											:= 1000.0 / (TIME_TO_LREAL(TimeImpImp));
	Forecast 												:= Forecast * (TIME_TO_REAL(Basetime) * 0.001);
	CountAct 												:= CountAct + 1;
	addNewPart												:= TRUE;
	Q_RT													:= TRUE;
END_METHOD

METHOD PUBLIC reset : bool //Return value = TRUE if execution finished
VAR_INPUT
END_VAR
	Forecast												:= 0;
	Counted													:= 0;
	CountAct												:= 0;
	reset													:= TRUE;
END_METHOD

END_FUNCTION_BLOCK

// ---- POUs/_Miscellaneous/64BitFunctions/CLEARBIT64.TcPOU
{attribute 'displaymode':='binary'}	
FUNCTION CLEARBIT64 : LWORD
VAR_INPUT
	inVal64			:	LWORD;
	bitNo			:	INT;
END_VAR
VAR
{attribute 'displaymode':='binary'}	
	lwConst 			:	LWORD := 1;
END_VAR

CLEARBIT64 := inVal64 AND NOT (SHL(lwConst,bitNo MOD 64));

END_FUNCTION

// ---- POUs/_Miscellaneous/nextIdx.TcPOU
FUNCTION nextIdx : BOOL //TRUE if incremented index is still in range
(* Example
	IF nextIdx(ActiveData, MIN_DATA,MAX_DATA)
	THEN
		State			:= State + 1; //continue to process next data set
	ELSE 
		State 			:= 99; //Done, no more data to process idx value will be = MAX_DATA
	END_IF
	
*)
VAR_IN_OUT
	idx					:	INT;
END_VAR
VAR_INPUT
	MinIdx				:	INT;
	MaxIdx				:	INT;
END_VAR
VAR
END_VAR

Idx 					:= MAX(MinIdx,Idx + 1);
IF Idx > MaxIdx
THEN
	idx					:= MaxIdx;
	nextIdx				:= FALSE;
ELSE
	nextIdx				:= TRUE;
END_IF

END_FUNCTION

// ---- POUs/_Miscellaneous/scale2.TcPOU
//Discription:	"SCALE" scales the In-Value, based on InLow to InHigh, to the commited OutLow and OutHigh ratio (In value will not be limited and Out values may exceed the given values according the exceed or undershot of In) 
//Used for AnalogIn/Out
FUNCTION scale2 : LREAL
VAR_INPUT
	In				 										: LREAL;
	InLow 													: LREAL;
	InHigh 													: LREAL;
	OutLow 													: LREAL;
	OutHigh 												: LREAL;
END_VAR
VAR
	Lim														: LREAL;
	X														: LREAL;
END_VAR

IF OutHigh <> OutLow 
THEN
	X														:= InHigh - InLow;
	IF x <> 0.0             									
	THEN       
		Lim 												:= In - InLow;             									
		X		 											:= (OutHigh - OutLow) / X;
		scale2 												:= (X * Lim) + OutLow;			
	ELSE                    									
		scale2												:= 0.0;
	END_IF
ELSE
	scale2													:= 0.0;	
END_IF

END_FUNCTION

// ---- POUs/_Miscellaneous/Conversions/ADSERROR_TO_HRESULT.TcPOU
{attribute 'no_check'}
//Convert ADS error id into HRESULT error enum
FUNCTION ADSERROR_TO_HRESULT : E_HRESULTAdsErr
VAR_INPUT
{attribute 'displaymode':='hex'}
	ErrorID													: UDINT;
END_VAR
VAR
END_VAR

IF ErrorID < 10000 //WS Error 
THEN	
	ADSERROR_TO_HRESULT				:= TO_DINT(ErrorID + TO_UDINT(16#98110000));
ELSIF ErrorID < TO_UDINT(16#98110000)
THEN
	ADSERROR_TO_HRESULT				:= E_HRESULTAdsErr.HRESULT_ADS_NOERROR;
ELSE
	ADSERROR_TO_HRESULT				:= TO_DINT(ErrorID); 
END_IF

END_FUNCTION

// ---- POUs/_Miscellaneous/Conversions/SWAP_WORDS_OF_DWORD.TcPOU
//Swaps high and low word of an DWORD variable
FUNCTION SWAP_WORDS_OF_DWORD : DWORD
VAR_INPUT
	in														:	DWORD;
END_VAR
VAR
	pTmp													:	POINTER TO WORD;
	WordArray												:	ARRAY[1..2] OF WORD;
	i														:	INT; 
END_VAR

	ptmp														:= ADR(In);
	WordArray[2]												:= ptmp^; // [1]
	ptmp														:= ptmp + 2;
	WordArray[1]												:= ptmp^; // [2]

	MEMCPY(ADR(SWAP_WORDS_OF_DWORD),ADR(WordArray),SIZEOF(WordArray));

END_FUNCTION

// ---- POUs/_Miscellaneous/Conversions/SWAP_WORDS_OF_LWORD.TcPOU
// Returns TRUE when words are successfully swapped 
FUNCTION SWAP_WORDS_OF_LWORD : LWORD
VAR_INPUT
	in														:	LWORD;
END_VAR
VAR
	pTmp													:	POINTER TO WORD;
	WordArray												:	ARRAY[1..4] OF WORD;
END_VAR

	pTmp													:= ADR(in);
	WordArray[4]											:= pTmp^; // [1]
	pTmp													:= pTmp + 2;
	WordArray[3]											:= pTmp^; // [2]
	pTmp													:= pTmp + 2;
	WordArray[2]											:= pTmp^; // [3]
	pTmp													:= pTmp + 2;
	WordArray[1]											:= pTmp^; // [4]
	
	Memcpy(ADR(SWAP_WORDS_OF_LWORD),ADR(WordArray),SIZEOF(WordArray));

END_FUNCTION

// ---- POUs/_Miscellaneous/CAM3D.TcPOU
{attribute 'monitoring' := 'variable'}
{attribute 'no_check'}
//if x,y,z in setpoint +/- window then cam3d = true else cam3d = false	
FUNCTION CAM3D : BOOL
VAR_INPUT
	X														: LREAL ;	//X-value to be monitored
	Y														: LREAL;	//Y-value to be monitored
	Z														: LREAL;	//Z-value to be monitored
	SETP_X													: LREAL ;	//X-target value
	SETP_Y													: LREAL ;	//Y-target value
	SETP_Z													: LREAL ;	//Z-target value
	WINDOW													: LREAL ;	//tolerance zone
END_VAR
VAR
END_VAR

	(* cam check				  											ds	*)
	(****************************************************************************)
	(* if x in setpoint +/- window then cam = true else cam = false				*)
	(****************************************************************************)

(* the current value of the window  *****************************************)
CAM3D 														:=  	X >= SETP_X - WINDOW AND X <= SETP_X + WINDOW
																AND Y >= SETP_Y - WINDOW AND Y <= SETP_Y + WINDOW
																AND Z >= SETP_Z - WINDOW AND Z <= SETP_Z + WINDOW;

(******************************************************************************)

END_FUNCTION

// ---- POUs/_Miscellaneous/polynomial.TcPOU
//calculate polynomial of certain degree
// y := p0 + p1*x^1 + p2*x^2 + p3*x^3 + p4*x^4 + p5*x^5 + p6*x^6 + p7*x^7 + p8*x^8;
FUNCTION polynomial : LREAL 							
VAR_INPUT
	X			: LREAL;
	Degree		: INT;

	p0			: LREAL;
	p1			: LREAL;
	p2			: LREAL;
	p3			: LREAL;
	p4			: LREAL;
	p5			: LREAL;
	p6			: LREAL;
	p7			: LREAL;
	p8			: LREAL;
END_VAR
VAR
END_VAR


IF degree >= 0 THEN Polynomial := 				p0 			  ; 	ELSE RETURN; END_IF
IF degree >= 1 THEN Polynomial := Polynomial + 	p1 * EXPT(x,1); 	ELSE RETURN; END_IF
IF degree >= 2 THEN Polynomial := Polynomial + 	p2 * EXPT(x,2); 	ELSE RETURN; END_IF
IF degree >= 3 THEN Polynomial := Polynomial + 	p3 * EXPT(x,3); 	ELSE RETURN; END_IF
IF degree >= 4 THEN Polynomial := Polynomial + 	p4 * EXPT(x,4); 	ELSE RETURN; END_IF
IF degree >= 5 THEN Polynomial := Polynomial + 	p5 * EXPT(x,5); 	ELSE RETURN; END_IF
IF degree >= 6 THEN Polynomial := Polynomial + 	p6 * EXPT(x,6); 	ELSE RETURN; END_IF
IF degree >= 7 THEN Polynomial := Polynomial + 	p7 * EXPT(x,7); 	ELSE RETURN; END_IF
IF degree >= 8 THEN Polynomial := Polynomial + 	p8 * EXPT(x,8); 	ELSE RETURN; END_IF

END_FUNCTION

// ---- POUs/_Miscellaneous/TOGGLE.TcPOU
{attribute 'no_check'}
//Toggle / FlipFlop
FUNCTION_BLOCK TOGGLE
VAR_INPUT
	IN														:	BOOL;
	RST														:	BOOL;
END_VAR             										
VAR_OUTPUT          										
	Q														:	BOOL;
END_VAR             	
VAR                 	
	M														:	BOOL;
END_VAR

	(* Toggle 				             	 																*)
	(************************************************************************************)

(* Ablauf ********************************************************************)
IF IN
	AND NOT M
THEN
	Q														:= NOT Q;
END_IF
M															:=	IN;
IF RST 
THEN 
	Reset(); 
END_IF


(********************************************************************************)

METHOD PUBLIC CLK : BOOL //Return value = status of output Q
VAR_INPUT
END_VAR
Q															:= NOT Q; 														
CLK 														:= Q;
END_METHOD

METHOD RESET : BOOL //Return value = TRUE if execution finished
VAR_INPUT
END_VAR
M := Q := FALSE;
RESET	:= TRUE;
END_METHOD

METHOD PUBLIC SET : BOOL  //Return value = TRUE if execution finished
VAR_INPUT
END_VAR
SET := M := Q := TRUE;
END_METHOD

END_FUNCTION_BLOCK

// ---- POUs/_Miscellaneous/WIN.TcPOU
{attribute 'monitoring' := 'variable'}
{attribute 'no_check'}
//if X between LO and HI then win = True else win = false
FUNCTION WIN : BOOL
VAR_INPUT
	X		: LREAL ;	
	LO		: LREAL ;
	HI		: LREAL ;
END_VAR
VAR
END_VAR

	(* window check 			  											ds	*)
	(****************************************************************************)
	(* if X between LO and HI then win = True else win = false					*)
	(****************************************************************************)


(* the current value of the window  *****************************************)
WIN 														:= 		X >= LO AND X <= HI;
(*****************************************************************************)

END_FUNCTION

// ---- POUs/Safety/Diag/SafetyIODeviceDiagRead.TcPOU
{attribute 'no_check'}
{attribute 'enable_dynamic_creation'}
FUNCTION_BLOCK SafetyIODeviceDiagRead EXTENDS FbBase
VAR CONSTANT
	bitTwinSAFETerm											:	BYTE := 0; //Ex1918,ELx9xx, etc. (2nd generation of TwinSAFE devices with CoE Index 10F3 Diag History included)
	bitSafetyTerm											:	BYTE := 1; //EL1904,EL2904,EK1914,EP1908 (Diagnoses provided via CoE Index 0x800E FSOE Internal Data, Debug 1..x) 
 	bitAX58xx												:	BYTE := 2; //AX5805,AX5806 (Diag via CoE index 0xFA10)
END_VAR
VAR_INPUT
	EcMasterDevId											:	UINT;	//EtherCAT Master DevId
END_VAR                 									
VAR_OUTPUT              									 
	AdsAddr											AT %I*	:	AMSADDR; //Link to terminal/box/device AMS Net Addr.
	{attribute 'displaymode':='binary'}
	MsgInfoDiag										AT %I*	:	USINT; 	//Link to connection messagediag of EL69xx (Needs to be enabled for alias of device)
//	{attribute 'displaymode':='hexadecimal'}
//	MsgInfoState									AT %I*	:	USINT; 	//Link to connection message state of EL69xx (Needs to be enabled for alias of device)	
	DevType													:	STRING(15); //CoE index 1008 / e.g. EL1908, EP1957-0022, etc...
	Name													:	STRING(31);	//Device name as defined in system manager configuration								
	FSoEAddr												:	WORD; //CoE index 0xF980
	DiagMsgSeverity											:	UINT; //Info (0) Warning (1) or Error (2)
	{attribute 'displaymode':='hexadecimal'}
	DiagMsgTextId											: 	UINT; //CoE Index 10F3 newest diagnoses message TextID (xyzz -> X =Type | y = Source | zz = Message ID)
	{attribute 'displaymode':='hexadecimal'}
	pDebugData												:	POINTER TO ARRAY[0..64] OF WORD; //Pointer to CoE index 0x800E - FSOE Internal Data - Debug 1-x for diag of "Safety Terminals" (or CoE Index 0xFA10 for AX58xx)
	DebugDataMaxId											:	UINT; //Max index for pointer pDebugData to array of word (Debug 1..x) if 0 data are invalid		
END_VAR                 									

VAR(* internal *)    
	{attribute 'displaymode':='bin'}
	DevCategory												:	BYTE;
	IOF_GetBoxNameByAddr									:	IOF_GetBoxNameByAddr := (TMOUT	:= DEFAULT_ADS_TIMEOUT);
	EcCoEReadDiagMsg										:	EcCoEReadNewestDiagMsg ;              									
	EcCoESdoReadEx											:	FB_EcCoESdoReadEx := (tTimeout := DEFAULT_ADS_TIMEOUT);       
	i														:	INT;  								                            	
END_VAR
(*
Tabelle 2-4: Diagnose-Informationen einer Connection
Wert Beschreibung
xxxx 0001 invalid command
xxxx 0010 unknown command
xxxx 0011 invalid connection ID
xxxx 0100 invalid CRC
xxxx 0101 Watchdog run out of time
xxxx 0110 invalid FSoE-Adress
xxxx 0111 invalid data
xxxx 1000 invalid length of communicatoin parameter Kommunikationsparameterlänge
xxxx 1001 invalid communicatoin parameter
xxxx 1010 invalid operator parameter length
xxxx 1011 invalid operator parameter
xxxx 1100 FSoE Master Reset
xxxx 1101 Module fault on slave detected with activated option "Modulfault is ComError"
xxxx 1110 Module fault on EL290x at activated with option "Error achnowledge active"
xxxx 1111 Slave not started or unexpected error argument

xxx1 xxxx FSoE Slave error detected
xx1x xxxx FSoE Slave notifies Failsafe Value active
x1xx xxxx StartUp
1xxx xxxx FSoE Master notifies Failsafe Value active
*)

(* IO Safety Terminal Status Diag		V2.0	*)
(************************************************)

(* Trigger to read diag **********************************************)
	rtExecute(CLK := Execute);
	
(* Read adress and type ***********************************************)
	CASE state OF
	0:
		Busy 												:= FALSE;
		IF NOT Execute
		THEN
			Done											:= FALSE;
			Error											:= FALSE;
			ErrorId											:= 0;					
		END_IF
		
		IF rtExecute.Q
		THEN
			Busy 											:= TRUE;
			Done											:= FALSE;
			Error											:= FALSE;
			ErrorId											:= 0;
			DiagMsgTextId									:= 0;
			DiagMsgSeverity									:= 0;

			EcCoESdoReadEx(bExecute := FALSE, bCompleteAccess := FALSE);
			IOF_GetBoxNameByAddr(Start := FALSE);
			EcCoEReadDiagMsg(Execute := FALSE);
			
			IF DevCategory.bitTwinSAFETerm
			THEN
				state 										:= 10;	
			ELSIF DevCategory.bitSafetyTerm
			THEN
				state 										:= SEL(DebugDataMaxId = 0, 21, 20);
			ELSIF DevCategory.bitAX58xx				
			THEN 
				state 										:= 30;
				
			ELSE //Read more device information 
				state										:= state + 1;				
			END_IF
		
		END_IF

	1: (* read FSOE adress *)
		EcCoESdoReadEx(
			sNetId			:= F_CreateAmsNetId(nIds := AdsAddr.netId ),
			nSlaveAddr		:= AdsAddr.port,
			nSubIndex		:= 16#1,
			nIndex			:= 16#F980,
			pDstBuf			:= ADR(FSOEAddr),
			cbBufLen		:= SIZEOF(FSOEAddr),
			bExecute		:= TRUE,
			tTimeout		:=  (* Default *),
			bCompleteAccess	:= False,
			bBusy			=> ,
			bError			=> ,
			nErrId			=> );
			
		IF NOT EcCoESdoReadEx.bBusy
		THEN
			IF EcCoESdoReadEx.bError 
			THEN
				Busy 										:= FALSE;
				Error										:= TRUE;
				ErrorId										:= EcCoESdoReadEx.nErrId;
				DiagMsgTextId								:= TO_UINT(state);
				state										:= 0;
			ELSE      									
				state 										:= state + 1;
			END_IF
			EcCoESdoReadEx(bExecute := FALSE);
		END_IF

	2: //Ready name from system manager configuration
		IOF_GetBoxNameByAddr(
			NETID		:='' , (* Local *)
			DEVICEID	:= UINT_TO_UDINT(EcMasterDevId) ,
			BOXADDR		:= AdsAddr.port ,
			START		:= EcMasterDevId <> 0,
			BOXNAME		=> );
			
		IF NOT IOF_GetBoxNameByAddr.Busy
		THEN
			IF IOF_GetBoxNameByAddr.Err 
			THEN
				Busy 										:= FALSE;
				Error										:= TRUE;
				ErrorId										:= IOF_GetBoxNameByAddr.ERRID;
				DiagMsgTextId								:= TO_UINT(state);
				state										:= 0;
			ELSIF IOF_GetBoxNameByAddr.Start
			THEN
				state 										:= state + 1;
			ELSE //No box name to read
				Name										:= CONCAT('EtherCAT Addr.',TO_STRING(AdsAddr.port));
			END_IF
			IOF_GetBoxNameByAddr(START := FALSE);
		END_IF
		
	3:  (* read device name e.g. EL1904 *)
		EcCoESdoReadEx(bExecute	:= TRUE, nIndex	:= 16#1008, nSubIndex := 16#0, pDstBuf := ADR(DevType),cbBufLen	:= SIZEOF(DevType), bCompleteAccess := FALSE);

		IF NOT EcCoESdoReadEx.bBusy
		THEN
			IF EcCoESdoReadEx.bError 
			THEN
				Busy 										:= FALSE;
				Error										:= TRUE;
				ErrorId										:= EcCoESdoReadEx.nErrId;
				DiagMsgTextId								:= TO_UINT(state);
				state										:= 0;
			ELSE       
				 //Delte type from name if in brakets 
				Name										:= DELETE(IOF_GetBoxNameByAddr.BOXNAME, LEN(DevType) + 2 , FIND(IOF_GetBoxNameByAddr.BOXNAME,DevType) - 1);
                             	
				IF DevType = 'AX5806' OR_ELSE DevType = 'AX5805'
				THEN
					DevCategory.bitAX58xx					:= TRUE;
					state 									:= 30;
				ELSIF DevType = 'EL1904' OR_ELSE DevType = 'EL2904' OR_ELSE DevType = 'EK1914' OR_ELSE DevType = 'EP1908'
				THEN
					DevCategory.bitSafetyTerm 				:= TRUE;
					state 									:= SEL(DebugDataMaxId = 0, 21, 20);
				ELSE
					DevCategory.bitTwinSAFETerm				:= TRUE;
					state 									:= 10;
				END_IF
				
			END_IF
			EcCoESdoReadEx(bExecute := FALSE);
		END_IF

	(* Read diagnoses latest entry from diag history ***********************************)	
	10: 
		EcCoEReadDiagMsg(Execute := TRUE, AdsAddr := AdsAddr);
		IF NOT EcCoEReadDiagMsg.Busy
		THEN
			IF EcCoEReadDiagMsg.Error 
			THEN
				Busy 										:= FALSE;
				Error										:= TRUE;
				ErrorId										:= EcCoEReadDiagMsg.ErrorID;
				DiagMsgTextId								:= TO_UINT(state);
				state										:= 0;				
			ELSE
				DiagMsgTextId								:= EcCoEReadDiagMsg.MsgId;
				DiagMsgSeverity								:= EcCoEReadDiagMsg.MsgSeverity;
				Done										:= TRUE;
				Busy										:= FALSE;
				State										:= 0;
			END_IF
		END_IF
		
	(* Read lenght of 0x800E:0 FSOE internal data.Debug terminal *********************************)
	20:
		EcCoESdoReadEx(bExecute	:= DebugDataMaxId = 0, nIndex	:= 16#800E, nSubIndex := 16#0, pDstBuf := ADR(DebugDataMaxId),cbBufLen	:= SIZEOF(DebugDataMaxId), bCompleteAccess := FALSE);

		IF NOT EcCoESdoReadEx.bBusy
		THEN
			IF EcCoESdoReadEx.bError 
			THEN
				Busy 										:= FALSE;
				Error										:= TRUE;
				ErrorId										:= EcCoESdoReadEx.nErrId;
				DiagMsgTextId								:= TO_UINT(state);
				state										:= 0;
			ELSIF DebugDataMaxId = 0
			THEN
				Busy 										:= FALSE;
				Error										:= TRUE;
				ErrorId										:= E_AdsErr.DEVICE_INVALIDPARM; //Lenght of index cannot be 0
				DiagMsgTextId								:= TO_UINT(state);
				state										:= 0;				
			ELSIF pDebugData = 0
			THEN                                  	
				pDebugData									:= __NEW(WORD,TO_UDINT(DebugDataMaxId + 1)); //e.g. 16 words = 32 bytes + 1 word for index 0 (which is in fact a byte  				
				IF PARAM.ENABLE_DEBUG_MSG_DYNAMIC_MEM_ALLOCATION
				THEN
					AdsLogHint('EngineeringToolbox | FB SafetyIOReadDiag | An instance allocated %s bytes from the dynamic memory of the ADS router memory pool', TO_STRING((DebugDataMaxId * 2) + 2));
				END_IF
				state 										:= state + 1;
			ELSE
				state 										:= state + 1;
			END_IF
			EcCoESdoReadEx(bExecute := FALSE);
		END_IF	
		
	21://Read all debug data from terminal
		EcCoESdoReadEx(bExecute	:= TRUE, nIndex	:= 16#800E, nSubIndex := 16#0, pDstBuf := pDebugData ,cbBufLen := TO_UDINT(DebugDataMaxId * 2) + SIZEOF(DebugDataMaxId) , bCompleteAccess := TRUE);

		IF NOT EcCoESdoReadEx.bBusy
		THEN
			IF EcCoESdoReadEx.bError 
			THEN
				IF pDebugData = 0
				THEN
					DebugDataMaxId							:= 0;
				END_IF
				Busy 										:= FALSE;
				Error										:= TRUE;
				ErrorId										:= EcCoESdoReadEx.nErrId;
				DiagMsgTextId								:= TO_UINT(state);
				state										:= 0;
			ELSE                                    		
				Done										:= TRUE;
				Busy										:= FALSE;
				DiagMsgSeverity								:= 2;
				State										:= 0;					
			END_IF
			EcCoESdoReadEx(bExecute := FALSE, bCompleteAccess := FALSE );
		END_IF			
	
	(* Read diag data from AX58xx *********************************)
	30:
		IF pDebugData = 0
		THEN
			DebugDataMaxId									:= 16#8;
			pDebugData										:= __NEW(WORD,TO_UDINT(DebugDataMaxId + 1));
			
			IF PARAM.ENABLE_DEBUG_MSG_DYNAMIC_MEM_ALLOCATION
			THEN
				AdsLogHint('EngineeringToolbox | FB SafetyIOReadDiag | An instance allocated %s bytes from the dynamic memory of the ADS router memory pool', '18');
			END_IF				
		END_IF
		
		EcCoESdoReadEx(bExecute	:= TRUE, nIndex	:= 16#FA10, nSubIndex := 16#0, pDstBuf := pDebugData, cbBufLen	:= TO_UDINT(DebugDataMaxId * 2) + SIZEOF(DebugDataMaxId),bCompleteAccess := TRUE);

		IF NOT EcCoESdoReadEx.bBusy
		THEN
			IF EcCoESdoReadEx.bError 
			THEN
				IF pDebugData = 0
				THEN
					DebugDataMaxId							:= 0;
				END_IF
				Busy 										:= FALSE;
				Error										:= TRUE;
				ErrorId										:= EcCoESdoReadEx.nErrId;
				DiagMsgTextId								:= TO_UINT(state);
				state										:= 0;
			ELSE                                    		
				Done										:= TRUE;
				Busy										:= FALSE;
				DiagMsgSeverity								:= 2;
				State										:= 0;	
			END_IF
			EcCoESdoReadEx(bExecute := FALSE, bCompleteAccess := FALSE);
		END_IF	
	ELSE
		;
	END_CASE
			
(*********************************************************************************************)

METHOD FB_exit : BOOL
VAR_INPUT
	bInCopyCode : BOOL; // if TRUE, the exit method is called for exiting an instance that is copied afterwards (online change).
END_VAR
IF NOT bInCopyCode AND pDebugData <> 0
THEN //Release memory in case the PLC stopps
	__DELETE(pDebugData);
	DebugDataMaxId								:= 0;
END_IF
END_METHOD

{attribute 'monitoring' := 'call'}
PROPERTY PUBLIC msgSevyIsError : BOOL
GET
msgSevyIsError := DiagMsgSeverity = 2;
END_GET
END_PROPERTY

{attribute 'monitoring' := 'call'}
PROPERTY PUBLIC msgSevyIsInfo : BOOL
GET
msgSevyIsInfo := DiagMsgSeverity = 0;
END_GET
END_PROPERTY

{attribute 'monitoring' := 'call'}
PROPERTY PUBLIC msgSevyIsWarning : BOOL
GET
msgSevyIsWarning := DiagMsgSeverity = 1;
END_GET
END_PROPERTY

END_FUNCTION_BLOCK

// ---- POUs/Safety/SafetyGroupIO.TcPOU
{attribute 'no_check'}
FUNCTION_BLOCK SafetyGroupIO
VAR_OUTPUT CONSTANT
//Group State
	STATE_UNKNOWN											: BYTE := 0;
	STATE_RUN												: BYTE := 1;
	STATE_STOP												: BYTE := 2;
	STATE_SAFE												: BYTE := 3; //Only EL6900
	STATE_ERROR												: BYTE := 4;
	STATE_RESET												: BYTE := 5;
	STATE_START												: BYTE := 6;
	STATE_STOP_ERROR										: BYTE := 7;
	STATE_DEACTIVE											: BYTE := 16;
	STATE_WAIT_COM_ERROR									: BYTE := 17; 
	
//Group Diag
	DIAG_OK													:	BYTE := 0;
	DIAG_FB_ERROR											:	BYTE := 1;
	DIAG_COM_ERROR											:	BYTE := 2;
	DIAG_MODULE_ERROR										:	BYTE := 3;
	DIAG_CMP_ERROR											:	BYTE := 4;
	DIAG_DEACTIVE_ERROR										:	BYTE := 5;
	DIAG_RESTART_ERROR										:	BYTE := 6;
END_VAR
VAR_INPUT
	ErrAck											AT  %Q*	:	BOOL := FALSE;	//Resets safety group error with rising edge 
	RunStop											AT  %Q* :	BOOL := TRUE;	//TRUE for run and FALSE for stop safety group 
	ModuleFault										AT  %Q* :	BOOL := FALSE;	//

END_VAR                     						
VAR_OUTPUT                  						
	ComErr											AT  %I* : 	BOOL;	//Safety group has a communication error
	ComStartup										AT  %I* :	BOOL;	//Only for EL6910
	FbDeactive										AT  %I* :	BOOL;	//Only for EL6910
	FBErr											AT  %I* : 	BOOL;	//Safety group has a FB error
	FbRun											AT  %I* :	BOOL;	//Only for EL6910
	InRun											AT  %I* :	BOOL;	//Only for EL6910
	OtherErr										AT  %I* :	BOOL;	//Only for EL6910
	OutErr											AT  %I* :	BOOL;	//Safety group has an output error
	
//Only available if the Checkboxes "MapState" and "MapDiag" are selected
	State											AT  %I* : USINT;	//Safety group state - 1=Run/2=Stop/3=Safe/4=Error/5=Reset
	Diag											AT  %I* : USINT;	//Safety group diagnostic information
END_VAR
VAR
END_VAR

(* SafetyGroup IO											             *)
(*************************************************************************)

(*************************************************************************)

{attribute 'monitoring' := 'call'}
PROPERTY Public diagCmpError : bool
GET
DiagCmpError:= Diag = DIAG_CMP_ERROR;
END_GET
END_PROPERTY

{attribute 'monitoring' := 'call'}
PROPERTY Public diagComError : bool
GET
DiagComError:= Diag = DIAG_COM_ERROR;
END_GET
END_PROPERTY

{attribute 'monitoring' := 'call'}
PROPERTY Public diagDeactiveError : bool
GET
DiagDeactiveError:= Diag = DIAG_DEACTIVE_ERROR;
END_GET
END_PROPERTY

{attribute 'monitoring' := 'call'}
PROPERTY PUBLIC diagFbError : BOOL
GET
DiagFbError:= Diag = DIAG_FB_ERROR;;
END_GET
END_PROPERTY

{attribute 'monitoring' := 'call'}
PROPERTY Public diagModuleError : bool
GET
DiagModuleError:= Diag = DIAG_MODULE_ERROR;
END_GET
END_PROPERTY

{attribute 'monitoring' := 'call'}
PROPERTY Public diagNoError : bool
GET
DiagNoError := Diag = 0;
END_GET
END_PROPERTY

{attribute 'monitoring' := 'call'}
PROPERTY Public diagRestartError : bool
GET
DiagRestartError:= Diag = DIAG_RESTART_ERROR;
END_GET
END_PROPERTY

{attribute 'monitoring' := 'call'}
PROPERTY PUBLIC inStateDeactive : bool
GET
inStateDeactive := State = STATE_DEACTIVE;
END_GET
END_PROPERTY

{attribute 'monitoring' := 'call'}
PROPERTY PUBLIC inStateError : BOOL
GET
inStateError :=	State = STATE_ERROR;
END_GET
END_PROPERTY

{attribute 'monitoring' := 'call'}
PROPERTY PUBLIC inStateReset : Bool
GET
inStateReset :=	State = STATE_RESET;
END_GET
END_PROPERTY

{attribute 'monitoring' := 'call'}
PROPERTY PUBLIC inStateRun : BOOL
GET
inStateRun :=	State = STATE_RUN;
END_GET
END_PROPERTY

{attribute 'monitoring' := 'call'}
PROPERTY PUBLIC inStateSafe : Bool
GET
inStateSafe :=	State = STATE_SAFE;
END_GET
END_PROPERTY

{attribute 'monitoring' := 'call'}
PROPERTY PUBLIC inStateStart : Bool
GET
inStateStart :=	State = STATE_START;
END_GET
END_PROPERTY

{attribute 'monitoring' := 'call'}
PROPERTY PUBLIC inStateStop : Bool
GET
inStateStop :=	State = STATE_STOP;
END_GET
END_PROPERTY

{attribute 'monitoring' := 'call'}
PROPERTY PUBLIC inStateStopError : bool
GET
inStateStopError := state = STATE_STOP_ERROR;
END_GET
END_PROPERTY

{attribute 'monitoring' := 'call'}
PROPERTY PUBLIC inStateUnknow : Bool
GET
inStateUnknow :=	State = STATE_UNKNOWN;
END_GET
END_PROPERTY

{attribute 'monitoring' := 'call'}
PROPERTY PUBLIC inStateWaitComError : bool
GET
inStateWaitComError := State = STATE_WAIT_COM_ERROR;
END_GET
END_PROPERTY

END_FUNCTION_BLOCK

// ---- POUs/Safety/SafetyPlcBackupRestore.TcPOU
{attribute 'no_check'}
FUNCTION_BLOCK SafetyPlcBackupRestore Extends FbBase
VAR_OUTPUT CONSTANT
	FNC_BACKUP_EXIST										:	INT := 0; //Check if backup file exists on hardware disk
	FNC_BACKUP												:	INT := 1; //Safe project on hardware disk as hex file
	FNC_RESTORE												:	INT := 2; //Write project back into EL69xx 
END_VAR             										
VAR_INPUT           										
	Fnc														:	INT (FNC_BACKUP_EXIST..FNC_RESTORE) := FNC_BACKUP;
	NetId													: 	T_AmsNetId := '';	//Net ID as text
	EcMasterNetID											: 	T_AmsNetId; 		//AmsNetID of the EtherCAT device *)
	EcMasterPort											: 	T_AmsPort; 			//Port Number of the EL6900 terminal (EtherCAT address) *)
	FilePath												:	T_MaxString := 'C:\'; //path to backup file
	FileName												:	STRING(20) := 'SafetyPlcFW.hex'; //name of backup file                      									
	Timeout													: 	TIME := T#60S;		//time until timeout
END_VAR
VAR_OUTPUT
	DataLength												:	UDINT := 0;
	ErrorFnc												:	STRING(30) := '';
END_VAR
VAR
(* Memory ***********************************************************)
	MemFnc													:	INT := -1;
	
(* Trigger **********************************************************)

(* Timer ************************************************************)
	tonDelay												:	ton;

(* blocks ***********************************************************)
	EnumFindFileEntry										:	FB_EnumFindFileEntry;
	BackupEL6900											:	FB_BackupEL6900;
	RestoreEL6900											:	FB_RestoreEL6900;
	
(* Dummys ***********************************************************)

END_VAR

	(************************************************************************************)
	(*																					*)
	(*		B E C K H O F F   N E W   A U T O M A T I O N   T E C H N O L O G Y    		*)
	(*																					*)
	(*		Eiserstr.5	D-33415 Verl	Germany	phone:	+49-5246-0	www.Beckhoff.Com	*)
    (*																					*)
    (*		Bausteinbeschreibung	:	Restore/Backup plc project 						*)
	(*		TwinCAT-Version			:	3.xx 											*)
	(*		Version					:	V1.1/ 05/16										*)
 	(*		Autor					:	Daniel Schlingmann								*)
	(*		Lib						:	tc2_backuprestoreel6900.compiled-library		*)
	(*																					*)
	(************************************************************************************)

(* Execute ***************************************************************************************)
	rtExecute(CLK := Execute);
	
	CASE state OF
	0:
		Busy												:= FALSE;
		// init		                                	
		IF NOT Execute                              	
		THEN        
			DataLength										:= 0;                                	
			Done 											:= FALSE;
			Error											:= FALSE;
			ErrorID											:= 0;
			ErrorFnc										:= '';
		END_IF                                      			                                            	
		IF rtExecute.Q                             	
		THEN                                        	
			Done 											:= FALSE;
			Busy											:= TRUE;
			Error											:= FALSE;
			ErrorID											:= 0;
			ErrorFnc										:= '';
			DataLength										:= 0;
			MemFnc											:= Fnc;
			BackupEL6900(ReadProject := FALSE);
			RestoreEL6900(writeProject := FALSE);
			EnumFindFileEntry(bExecute := FALSE, sNetId := '', tTimeout := Timeout, sPathName := CONCAT(FilePath,FileName));
			CASE Fnc OF
			FNC_BACKUP_EXIST:state							:= 1;		
			FNC_BACKUP		:state							:= 10;									
			FNC_RESTORE		:state							:= 20;									
			ELSE
				Busy										:= FALSE;
				Done										:= FALSE;
				Error										:= TRUE;
				ErrorId										:= E_AdsErr.DEVICE_INVALIDPARM;	
				ErrorFnc									:= 'SafetyPlcBackupRestore';					
			END_CASE
		END_IF
	
	(* Backup exists *****************************************************)
	1: //first abort old command
		EnumFindFileEntry(bExecute := TRUE ,eCmd := eEnumCmd_Abort );
		IF NOT EnumFindFileEntry.bBusy
		THEN
			EnumFindFileEntry(bExecute := FALSE ,eCmd := eEnumCmd_Abort );
			EnumFindFileEntry(bExecute := TRUE ,eCmd := eEnumCmd_First );
			state											:= State + 1;
		END_IF

	2: //read entrys
		EnumFindFileEntry(bExecute := TRUE);
		IF NOT EnumFindFileEntry.bBusy
		THEN
			IF NOT EnumFindFileEntry.bError
				AND EnumFindFileEntry.stFindFile.sFileName = FileName
			THEN
				Done										:= TRUE;
				Busy										:= FALSE;
				DataLength 									:= EnumFindFileEntry.stFindFile.fileSize.dwLowPart;
				state										:= 0;
			ELSE
				Busy										:= FALSE;
				Done										:= FALSE;
				Error										:= TRUE;
				ErrorId										:= SEL(EnumFindFileEntry.bError , E_AdsErr.DEVICE_NOTFOUND ,EnumFindFileEntry.nErrID);
				ErrorFnc									:= 'EnumFindFileEntry';
				state										:= 0;
			END_IF		
		END_IF
		
	(* Backup (save project to disk) *************************************************************)
	10:
		IF NOT BackupEL6900.bBusy
		THEN
			BackupEL6900(
				ReadProject		:= TRUE, 
				EtherCATAmsNetID:= EcMasterNetID, 
				Port			:= EcMasterPort, 
				FileWriteAmsNetID:= '', 
				FilePathname	:= CONCAT(FilePath,FileName), 
				bBusy			=> , 
				bError			=> , 
				uErrID			=> , 
				ReadDataLength	=> );
			state											:= state + 1;	
		ELSE
			BackupEL6900(ReadProject := FALSE);
		END_IF
		
	11:
		BackupEL6900();
		IF NOT BackupEL6900.bBusy
		THEN
			IF BackupEL6900.bError
			THEN
				Busy										:= FALSE;
				Done										:= FALSE;
				Error										:= TRUE;
				ErrorId										:= BackupEL6900.uErrID;
				ErrorFnc									:= 'BackupEL6900';
				state										:= 0;				
			ELSE
				Done										:= TRUE;
				Busy										:= FALSE;
				DataLength 									:= BackupEL6900.ReadDataLength;	
				state										:= 0;			
			END_IF
		END_IF

	(* Restore *************************************************************)
	20:
		IF NOT RestoreEL6900.bBusy
		THEN
			RestoreEL6900(
				WriteProject	:= TRUE, 
				EtherCATAmsNetID:= EcMasterNetID, 
				Port			:= EcMasterPort, 
				FileReadAmsNetID:= '', 
				FilePathname	:= CONCAT(FilePath,FileName), 
				bBusy			=> , 
				bError			=> , 
				uErrID			=> , 
				WriteDataLength	=> );
			state											:= state + 1;	
		ELSE
			RestoreEL6900(WriteProject := FALSE);
		END_IF
		
	21:
		RestoreEL6900();
		IF NOT RestoreEL6900.bBusy
		THEN
			IF RestoreEL6900.bError
			THEN
				Busy										:= FALSE;
				Done										:= FALSE;
				Error										:= TRUE;
				ErrorId										:= RestoreEL6900.uErrID;
				ErrorFnc									:= 'RestoreEL6900';
				state										:= 0;				
			ELSE
				Done										:= TRUE;
				Busy										:= FALSE;
				DataLength 									:= RestoreEL6900.WriteDataLength;	
				state										:= 0;			
			END_IF
		END_IF
		
	END_CASE
			
(*************************************************************************************************)

METHOD PUBLIC backup : BOOL //Return value = TRUE if busy
//required parameter
//EcMasterNetID
//EcMasterPort
//FilePath
VAR_INPUT
	Execute													:	BOOL;
END_VAR
CASE state OF
0:	
	Fnc 													:= FNC_BACKUP;
	THIS^(Execute:=Execute);
1: 
	;

END_CASE
Backup 														:= Busy;
END_METHOD

METHOD PUBLIC fileExists : BOOL //Return value = TRUE if busy
//required parameter
//FilePath
VAR_INPUT
	Execute													:	BOOL;
END_VAR
CASE state OF
0:	
	Fnc 													:= FNC_BACKUP_EXIST;
	THIS^(Execute:=Execute);
1: 
	;

END_CASE
fileExists 														:= Busy;
END_METHOD

METHOD PUBLIC restore : BOOL //Return value = TRUE if busy
//required parameter
//EcMasterNetID
//EcMasterPort
//FilePath
VAR_INPUT
	Execute													:	BOOL;
END_VAR
CASE state OF
0:	
	Fnc 													:= FNC_RESTORE;
	THIS^(Execute:=Execute);
1: 
	;

END_CASE
Restore 													:= Busy;
END_METHOD

END_FUNCTION_BLOCK

// ---- POUs/Motion/TF50xx-NC/02_Options/Motion/AxSuperposition.TcPOU
FUNCTION_BLOCK AxSuperposition EXTENDS AxFbBase
VAR_OUTPUT CONSTANT 
	FNC_MOVEIMPOSED											:	INT := 0;
	FNC_MOVEABORT											:	INT := 1;
END_VAR                     								
VAR_INPUT                   								
	Fnc														:	INT := FNC_MOVEIMPOSED;
	Mode    												:	E_SuperpositionMode;
	Distance      											:	LREAL;
	VelocityDiff 											:	LREAL;
	Acc			 											:	LREAL;
	Dec			 											:	LREAL;
	Jerk    												:	LREAL;
	VelocityProcess   										:	LREAL;
	Length    												:	LREAL;
	Options    												:	ST_SuperpositionOptions;
                            							
END_VAR
VAR_IN_OUT
END_VAR
VAR_OUTPUT
	Warning													:	BOOL;
	WarningId												:	UDINT;
END_VAR
VAR
(* Zwischenspeicher ****************************************)
	MemFnc													:	INT := -1;

(* Timer ***************************************************)

(* Trigger *************************************************)

(* Instanzierung der MC Bausteine **************************)
	MC_MoveImposed											:	MC_MoveSuperImposed;
	MC_MoveAbort											:	MC_AbortSuperposition;

(* Dummy Speicher ******************************************)

END_VAR

	(************************************************************************************)
	(*																					*)
	(*		B E C K H O F F   N E W   A U T O M A T I O N   T E C H N O L O G Y    		*)
	(*																					*)
	(*		Eiserstr.5	D-33415 Verl	Germany	phone:	+49-5246-0	www.Beckhoff.com	*)
  	(*																					*)
  	(*		Bausteinbeschreibung	:	Move Imposed Achs Baustein						*)
	(*		TwinCAT-Version			:	3.1		 										*)
	(*		Version					:	V1.0 / 04/16									*)
 	(*																					*)
	(*																					*)
	(************************************************************************************)

(* Execute ******************************************************************************)
	rtExecute(CLK := Execute);
	IF rtExecute.Q
		AND MemFnc < 0
	THEN
		MemFnc 												:= Fnc ;
		Busy												:= TRUE;
		Done												:= FALSE;
		Active												:= FALSE;
		Error												:= FALSE;
		ErrorID												:= 0;
		Warning												:= FALSE;
		WarningId											:= 0;
		CmdAborted											:= FALSE;
		ErrorText											:= '';
	END_IF

(* Call Method ***********************************************************************************)
	CASE MemFnc OF
	FNC_MOVEIMPOSED:
		MoveImposed(Execute);

	FNC_MOVEABORT:
		MoveAbort(Execute);

	-1:
		IF NOT Execute
		THEN
			Busy											:= FALSE;
			Done											:= FALSE;
			Active											:= FALSE;
			Error											:= FALSE;
			ErrorID											:= 0;
			Warning											:= FALSE;
			WarningId										:= 0;
			CmdAborted										:= FALSE;
			ErrorText										:= '';
		END_IF
	ELSE
		Busy												:= FALSE;
		Done												:= FALSE;
		Active												:= FALSE;
		Error												:= Execute;
		ErrorID												:= E_AdsErr.DEVICE_INVALIDPARM;
		Warning												:= Execute;
		WarningId											:= 0;
		CmdAborted											:= FALSE;
		ErrorText											:= CONCAT('invalid parameter value(s) Fnc no: ' , INT_TO_STRING(MemFnc));
	END_CASE

(*************************************************************************************************)

METHOD PUBLIC moveAbort : BOOL //Return value = TRUE if busy
VAR_INPUT
	Execute													:	BOOL;
END_VAR
	MemFnc 													:= FNC_MOVEABORT;

IF NOT __ISVALIDREF(rAxis) 
THEN
	Busy													:= NOT Error;
	Error													:= TRUE;
	ErrorId													:= E_AdsErr.DEVICE_INVALIDPARM;
	CmdAborted												:= FALSE;
	Done													:= FALSE;
	Active													:= FALSE;
	ErrorText												:= 'Reference rAxis invalid (0)';
	MemFnc													:= SEL(Execute , -1 ,MemFnc); 
	RETURN;
END_IF


MC_MoveAbort(
	Execute													:= Execute,
	Axis													:= rAxis,
	Done													=> Done,
	Busy													=> Busy,
	Error													=> Error,
	ErrorID													=> ErrorID);

	IF Error THEN
		LastErrorId											:= ErrorID;
		ErrorText 											:= CONCAT('Error MC_MoveAbort ID:' , UDINT_TO_STRING(ErrorId));
	ELSE
		ErrorText 											:= '';
	END_IF

	IF NOT Execute AND NOT Busy
	THEN
		MemFnc												:=  -1;
	END_IF

	MoveAbort												:= Busy;
END_METHOD

METHOD PUBLIC moveImposed : BOOL //Return value = TRUE if busy
VAR_INPUT
	Execute													:	BOOL;
END_VAR
	MemFnc 													:= FNC_MOVEIMPOSED;
	
IF NOT __ISVALIDREF(rAxis) 
THEN
	Busy													:= NOT Error;
	Error													:= TRUE;
	ErrorId													:= E_AdsErr.DEVICE_INVALIDPARM;
	CmdAborted												:= FALSE;
	Done													:= FALSE;
	Active													:= FALSE;
	ErrorText												:= 'Reference rAxis invalid (0)';
	MemFnc													:= SEL(Execute , -1 ,MemFnc); 
	RETURN;
END_IF

	MC_MoveImposed(
		Execute												:= Execute,
		Mode												:= Mode,
		Distance											:= Distance,
		VelocityDiff										:= VelocityDiff,
		Acceleration										:= Acc,
		Deceleration										:= Dec,
		Jerk												:= Jerk,
		VelocityProcess										:= VelocityProcess,
		Length												:= Length,
		Options												:= Options,
		Axis												:= rAxis,
		Done												=> Done,
		Busy												=> Busy,
		Active												=> Active,
		CommandAborted										=> CmdAborted,
		Error												=> Error,
		ErrorID												=> ErrorID,
		Warning												=> Warning,
		WarningId											=> WarningID,
		ActualVelocityDiff									=> ,
		ActualDistance										=> ,
		ActualLength										=> ,
		ActualAcceleration									=> ,
		ActualDeceleration									=> );


	IF Error THEN
		LastErrorId											:= ErrorID;
		ErrorText 											:= CONCAT('Error MC_MoveSuperImposed ID:' , UDINT_TO_STRING(ErrorId));
	ELSE                            					
		ErrorText 											:= '';
	END_IF

	IF NOT Execute AND NOT Busy
	THEN
		MemFnc												:=  -1;
	END_IF

	MoveImposed												:= Busy;
END_METHOD

END_FUNCTION_BLOCK

// ---- POUs/Motion/TF5100-NCI/02_Options/PlcItp/NciCreateItpTable.TcPOU
{attribute 'no_check'}
//Create Nci PlcInterpolation tabel
//
FUNCTION_BLOCK NciCreateItpTable
VAR_INPUT
	BlockNo													: UDINT := 0; //Block number addtional parameter for methods. At 0 -> block number will be automatically increased by every new entry
	OffsetFactorTblNumber									: UDINT := 100; 
	MaxTblNumber											: UDINT := 1000; 
END_VAR                     								
VAR_OUTPUT                  								
	Table													: ST_NciFeedGroupTable;
	FilledRows												: INT;
	LastBlockNo												: UDINT; //Last Blocknumber 
	Error													: BOOL;
{attribute 'displaymode':='hex'}
	ErrorID													: UDINT;
	ErrorText												: STRING(20);
END_VAR                     								
VAR
// Cache *******************************************
	TableNumber												: UDINT := 0;
	BlockCount												: UDINT := 1;

// Timer ******************************************************
// Trigger ****************************************************
// Blocks *****************************************************
	TblTemplate												: NciCreateItpTableEntryTemplate;
// Error ******************************************************
// Dummy Speicher *********************************************
	i														: INT := 0;
END_VAR

(* writing TcPlcInterpolation table				V1.5	*)
(********************************************************)

(* pleas use methods instead of the function-block body ********************)
	;
(***************************************************************************)

METHOD addCircleCIP : BOOL //Return value = TRUE if executed succesful
VAR_INPUT
	X														: LREAL := 0.0;
	Y														: LREAL := 0.0;
	Z														: LREAL := 0.0;
	Q1														: LREAL := 0.0;
	Q2														: LREAL := 0.0;
	Q3														: LREAL := 0.0;
	Q4														: LREAL := 0.0;
	Q5														: LREAL := 0.0;
	Velo													: LREAL; 	// mm/s 
	AccurateStop											: BOOL := FALSE;
	CIPPosX													: LREAL := 0.0;
	CIPPosY													: LREAL := 0.0;
	CIPPosZ													: LREAL := 0.0;
END_VAR
	(* NCI GeoCirclePlane schreiben									*)
	(*********************************************************)

(* Zielpos. in Tabelle schreiben ************************************************************)
	BlockCount 												:= BlockCount + 1;
	TblTemplate.GeoCircleCIP.nDisplayIndex := LastBlockNo 	:= SEL(BlockNo = 0, BlockNo, TableNumber * OffsetFactorTblNumber + BlockCount);
	TblTemplate.GeoCircleCIP.fEndPosX						:= X;
	TblTemplate.GeoCircleCIP.fEndPosY						:= Y;
	TblTemplate.GeoCircleCIP.fEndPosZ						:= Z;
	TblTemplate.GeoCircleCIP.fEndPosQ1						:= Q1;
	TblTemplate.GeoCircleCIP.fEndPosQ2						:= Q2;
	TblTemplate.GeoCircleCIP.fEndPosQ3						:= Q3;
	TblTemplate.GeoCircleCIP.fEndPosQ4						:= Q4;
	TblTemplate.GeoCircleCIP.fEndPosQ5						:= Q5;
	TblTemplate.GeoCircleCIP.fVelo							:= Velo;
	TblTemplate.GeoCircleCIP.bAccurateStop					:= AccurateStop;
	TblTemplate.GeoCircleCIP.fCIPPosX						:= CIPPosX;
	TblTemplate.GeoCircleCIP.fCIPPosY						:= CIPPosY;
	TblTemplate.GeoCircleCIP.fCIPPosZ						:= CIPPosZ;
                                                        	
	TblTemplate.InsertGeoCircleCIP(Table:= Table);    	
	Error													:= TblTemplate.Error;
	ErrorId													:= TblTemplate.ErrorId;
	ErrorText												:= TblTemplate.ErrorText;
	FilledRows												:= TblTemplate.FilledRows;

	AddCircleCip											:= NOT Error;
(***************************************************************************)
END_METHOD

METHOD addDwellTime : BOOL //Return value = TRUE if executed succesful
VAR_INPUT
	/// UCS ObjectID 
	Value													: LREAL ;
END_VAR
(*  													*)
(********************************************************)
	BlockCount 												:= BlockCount + 1;
	TblTemplate.DwellTime.nDisplayIndex	 := LastBlockNo 	:= SEL(BlockNo = 0, BlockNo, TableNumber * OffsetFactorTblNumber + BlockCount);
	TblTemplate.DwellTime.fDwellTime						:= Value;

	TblTemplate.InsertDwellTime(Table:= Table);
	Error													:= TblTemplate.Error;
	ErrorId													:= TblTemplate.ErrorId;
	ErrorText												:= TblTemplate.ErrorText;
	FilledRows												:= TblTemplate.FilledRows;

	AddDwellTime											:= not Error;	
	

(***************************************************************************)
END_METHOD

METHOD addEndOfTable : BOOL //Return value = TRUE if executed succesful
TblTemplate.InsertEndOfTable(Table:= Table);
Error													:= TblTemplate.Error;
ErrorId													:= TblTemplate.ErrorId;
ErrorText												:= TblTemplate.ErrorText;
FilledRows												:= TblTemplate.FilledRows;

AddEndOfTable											:= NOT Error;
END_METHOD

METHOD addMFuncFast : BOOL //Return value = TRUE if executed succesful
VAR_INPUT
	MFuncNo													: INT := 0;
END_VAR
(*														*)
(********************************************************)

(*************************************************************************************)
	BlockCount 												:= BlockCount + 1;
	TblTemplate.MFuncFast.nDisplayIndex := LastBlockNo 		:= SEL(BlockNo = 0, BlockNo, TableNumber * OffsetFactorTblNumber + BlockCount);
	TblTemplate.MFuncFast.nMFuncIn0							:= MFuncNo;
	TblTemplate.MFuncFast.nMFuncIn1							:= -1;
	TblTemplate.MFuncFast.nMFuncIn2							:= -1;
	TblTemplate.MFuncFast.nMFuncIn3							:= -1;
	TblTemplate.MFuncFast.nMFuncIn4							:= -1;
	TblTemplate.MFuncFast.nMFuncIn5							:= -1;
	TblTemplate.MFuncFast.nMFuncIn6							:= -1;
	TblTemplate.MFuncFast.nMFuncIn7							:= -1;
	
	TblTemplate.InsertMFuncFast(Table:= Table);
	Error													:= TblTemplate.Error;
	ErrorId													:= TblTemplate.ErrorId;
	ErrorText												:= TblTemplate.ErrorText;
	FilledRows												:= TblTemplate.FilledRows;
	
	AddMFuncFast											:= not Error;
(*************************************************************************************)
END_METHOD

METHOD addMFuncFastList : BOOL //Return value = TRUE if executed succesful
VAR_INPUT
	MFuncNo0												: INT := -1; //0-159 > Set to -1 to mark end of used MFunc
	MFuncNo1												: INT := -1; //0-159 > Set to -1 to mark end of used MFunc
	MFuncNo2												: INT := -1; //0-159 > Set to -1 to mark end of used MFunc
	MFuncNo3												: INT := -1; //0-159 > Set to -1 to mark end of used MFunc
	MFuncNo4												: INT := -1; //0-159 > Set to -1 to mark end of used MFunc
	MFuncNo5												: INT := -1; //0-159 > Set to -1 to mark end of used MFunc
	MFuncNo6												: INT := -1; //0-159 > Set to -1 to mark end of used MFunc
	MFuncNo7												: INT := -1; //0-159 > Set to -1 to mark end of used MFunc
END_VAR
(*														*)
(********************************************************)

(*************************************************************************************)
	BlockCount 												:= BlockCount + 1;
	TblTemplate.MFuncFast.nDisplayIndex := LastBlockNo 		:= SEL(BlockNo = 0, BlockNo, TableNumber * OffsetFactorTblNumber + BlockCount);
	TblTemplate.MFuncFast.nMFuncIn0							:= MFuncNo0;
	TblTemplate.MFuncFast.nMFuncIn1							:= MFuncNo1;
	TblTemplate.MFuncFast.nMFuncIn2							:= MFuncNo2;
	TblTemplate.MFuncFast.nMFuncIn3							:= MFuncNo3;
	TblTemplate.MFuncFast.nMFuncIn4							:= MFuncNo4;
	TblTemplate.MFuncFast.nMFuncIn5							:= MFuncNo5;
	TblTemplate.MFuncFast.nMFuncIn6							:= MFuncNo6;
	TblTemplate.MFuncFast.nMFuncIn7							:= MFuncNo7;
	
	TblTemplate.InsertMFuncFast(Table:= Table);
	Error													:= TblTemplate.Error;
	ErrorId													:= TblTemplate.ErrorId;
	ErrorText												:= TblTemplate.ErrorText;
	FilledRows												:= TblTemplate.FilledRows;
	
	AddMFuncFastList										:= NOT Error;
(*************************************************************************************)
END_METHOD

METHOD addMFuncHsk : BOOL //Return value = TRUE if executed succesful
VAR_INPUT
	MFuncNo													: INT := 0;
END_VAR
(* 														*)
(********************************************************)

(*************************************************************************************)
	BlockCount 												:= BlockCount + 1;
	TblTemplate.MFuncHsk.nDisplayIndex := LastBlockNo 		:= SEL(BlockNo = 0, BlockNo,  TableNumber * OffsetFactorTblNumber + BlockCount);
	TblTemplate.MFuncHsk.nMFunc								:= MFuncNo;
                                                        	
	TblTemplate.InsertMFuncHsk(Table:= Table);          	
	Error													:= TblTemplate.Error;
	ErrorId													:= TblTemplate.ErrorId;
	ErrorText												:= TblTemplate.ErrorText;
	FilledRows												:= TblTemplate.FilledRows;
	
	AddMFuncHsk												:= not Error;
(*************************************************************************************)
END_METHOD

METHOD addMFuncResetAllFast : BOOL //Return value = TRUE if executed succesful
VAR_INPUT
END_VAR
(* NCI ResetAllFastMFunc schreiben								*)
(*************************************************************************************)

(* confirmError all fast M-functions****************************************************)
	BlockCount 													:= BlockCount + 1;
	TblTemplate.MFuncResetAllFast.nDisplayIndex	:= LastBlockNo 	:= SEL(BlockNo = 0, BlockNo, TableNumber * OffsetFactorTblNumber + BlockCount);
	TblTemplate.InsertMFuncResetAllFast(Table:= Table);
	Error														:= TblTemplate.Error;
	ErrorId														:= TblTemplate.ErrorId;
	ErrorText													:= TblTemplate.ErrorText;
	FilledRows													:= TblTemplate.FilledRows;
	
	AddMFuncResetAllFast										:= not Error;
(*************************************************************************************)
END_METHOD

METHOD reset : BOOL //Return value = TRUE if execution finished
VAR_INPUT
END_VAR
TblTemplate.Reset(Table := Table);
FilledRows													:= 0;
BlockCount 													:= 0;
LastBlockNo													:= 0;
TableNumber 												:= TableNumber + 1;

IF TableNumber > MaxTblNumber 
THEN 
	TableNumber 											:= 1; 
END_IF

Error 														:= FALSE;
Errorid														:= 0;
ErrorText													:= '';
Reset														:= TRUE;
END_METHOD

METHOD setAxisDynamics : bool //Return value = TRUE if executed succesful
VAR_INPUT
	AxisNo													:	UDINT;
	Acc,Dec,Jerk											:	LREAL;
END_VAR
	(* NCI SetAxisDynamics schreiben						*)
	(*********************************************************)

(* Zielpos. in Tabelle schreiben ************************************************************)
	BlockCount 												:= BlockCount + 1;
	TblTemplate.AxisDynamics.nDisplayIndex := LastBlockNo := SEL(BlockNo = 0, BlockNo, TableNumber * OffsetFactorTblNumber + BlockCount);

	TblTemplate.AxisDynamics.nAxis 							:= AxisNo;
	TblTemplate.AxisDynamics.fDec							:= Dec;
	TblTemplate.AxisDynamics.fJerk							:= Jerk;
	TblTemplate.AxisDynamics.fAcc							:= Acc;
                                                        	
	TblTemplate.InsertAxisDynamics(Table:= Table);    	
	Error													:= TblTemplate.Error;
	ErrorId													:= TblTemplate.ErrorId;
	ErrorText												:= TblTemplate.ErrorText;
	FilledRows												:= TblTemplate.FilledRows;

	SetAxisDynamics											:= NOT Error;
(***************************************************************************)
END_METHOD

METHOD setBaseFrame : bool //Return value = TRUE if executed succesful
VAR_INPUT
    ShiftX													: LREAL;
    ShiftY													: LREAL;
    ShiftZ													: LREAL;
    RotX													: LREAL;
    RotY													: LREAL;
    RotZ													: LREAL;
    ShiftQ1													: LREAL;
    ShiftQ2													: LREAL;
    ShiftQ3													: LREAL;
    ShiftQ4													: LREAL;
    ShiftQ5													: LREAL;
END_VAR
	(* NCI SetBaseFrame schreiben						*)
	(*********************************************************)

(* Zielpos. in Tabelle schreiben ************************************************************)
	BlockCount 												:= BlockCount + 1;
	TblTemplate.BaseFrame.nDisplayIndex := LastBlockNo := SEL(BlockNo = 0, BlockNo, TableNumber * OffsetFactorTblNumber + BlockCount);

    TblTemplate.BaseFrame.fShiftX 							:= ShiftX;
    TblTemplate.BaseFrame.fShiftY							:= ShiftY;
    TblTemplate.BaseFrame.fShiftZ							:= ShiftZ;
    TblTemplate.BaseFrame.fRotX								:= RotX;
    TblTemplate.BaseFrame.fRotY								:= RotY;
    TblTemplate.BaseFrame.fRotZ								:= RotZ;
    TblTemplate.BaseFrame.fShiftQ1							:= ShiftQ1;
    TblTemplate.BaseFrame.fShiftQ2							:= ShiftQ2;
    TblTemplate.BaseFrame.fShiftQ3							:= ShiftQ3;
    TblTemplate.BaseFrame.fShiftQ4							:= ShiftQ4;
    TblTemplate.BaseFrame.fShiftQ5							:= ShiftQ5;
                       	
	TblTemplate.InsertBaseFrame(Table:= Table);    	
	Error													:= TblTemplate.Error;
	ErrorId													:= TblTemplate.ErrorId;
	ErrorText												:= TblTemplate.ErrorText;
	FilledRows												:= TblTemplate.FilledRows;

	SetBaseFrame											:= NOT Error;
(***************************************************************************)
END_METHOD

